LIN {X 0,Y 355.498,Z 368.258,A -85,B 0,C 180,E1 -13423.14,E2 -13423.14} C_VEL
LIN {X 0,Y 356.575,Z 358.586,A -85,B 0,C 180,E1 -13424.845,E2 -13424.845} C_VEL
LIN {X 0,Y 357.7,Z 348.667,A -85,B 0,C 180,E1 -13426.258,E2 -13426.258} C_VEL
LIN {X 0,Y 359.05,Z 337.613,A -85,B 0,C 180,E1 -13427.513,E2 -13427.513} C_VEL
LIN {X 0,Y 359.817,Z 328.864,A -85,B 0,C 180,E1 -13428.335,E2 -13428.335} C_VEL
LIN {X 0,Y 359.129,Z 316.785,A -85,B 0,C 180,E1 -13429.331,E2 -13429.331} C_VEL
LIN {X 0,Y 357.275,Z 303.493,A -85,B 0,C 180,E1 -13430.237,E2 -13430.237} C_VEL
LIN {X 0,Y 354.783,Z 291.013,A -85,B 0,C 180,E1 -13430.922,E2 -13430.922} C_VEL
LIN {X 0,Y 354.186,Z 288.154,A -85,B 0,C 180,E1 -13431.077,E2 -13431.077} C_VEL
LIN {X 0,Y 354.706,Z 281.188,A -85,B 0,C 180,E1 -13434.586,E2 -13434.586} C_VEL
LIN {X 0,Y 355.351,Z 273.981,A -85,B 0,C 180,E1 -13438.336,E2 -13438.336} C_VEL
LIN {X 0,Y 356.313,Z 266.953,A -85,B 0,C 180,E1 -13442.177,E2 -13442.177} C_VEL
LIN {X 0,Y 357.117,Z 261.205,A -85,B 0,C 180,E1 -13445.488,E2 -13445.488} C_VEL
LIN {X 0,Y 357.179,Z 257.764,A -85,B 0,C 180,E1 -13447.586,E2 -13447.586} C_VEL
LIN {X 0,Y 356.457,Z 253.353,A -85,B 0,C 180,E1 -13450.588,E2 -13450.588} C_VEL
LIN {X 0,Y 355.653,Z 249.108,A -85,B 0,C 180,E1 -13453.757,E2 -13453.757} C_VEL
LIN {X 0,Y 354.818,Z 244.397,A -85,B 0,C 180,E1 -13457.664,E2 -13457.664} C_VEL
LIN {X 0,Y 354.814,Z 244.29,A -85,B 0,C 180,E1 -13460.664,E2 -13460.664} C_VEL
LIN {X 0,Y 354.821,Z 244.29,A -85,B 0,C 180,E1 -13464.299,E2 -13464.299} C_VEL
LIN {X 0,Y 354.785,Z 244.294,A -85,B 0,C 180,E1 -13467.665,E2 -13467.665} C_VEL
LIN {X 0,Y 354.867,Z 244.283,A -85,B 0,C 180,E1 -13470.62,E2 -13470.62} C_VEL
LIN {X 0,Y 354.896,Z 244.279,A -85,B 0,C 180,E1 -13474.171,E2 -13474.171} C_VEL
LIN {X 0,Y 354.831,Z 244.287,A -85,B 0,C 180,E1 -13477.892,E2 -13477.892} C_VEL
LIN {X 0,Y 354.919,Z 244.276,A -85,B 0,C 180,E1 -13481.889,E2 -13481.889} C_VEL
LIN {X 0,Y 354.939,Z 244.273,A -85,B 0,C 180,E1 -13485.979,E2 -13485.979} C_VEL
LIN {X 0,Y 354.978,Z 244.269,A -85,B 0,C 180,E1 -13489.734,E2 -13489.734} C_VEL
LIN {X 0,Y 355.109,Z 244.253,A -85,B 0,C 180,E1 -13492.035,E2 -13492.035} C_VEL
LIN {X 0,Y 355.088,Z 244.255,A -85,B 0,C 180,E1 -13494.319,E2 -13494.319} C_VEL
LIN {X 0,Y 355.24,Z 244.237,A -85,B 0,C 180,E1 -13497.731,E2 -13497.731} C_VEL
LIN {X 0,Y 355.391,Z 244.218,A -85,B 0,C 180,E1 -13499.998,E2 -13499.998} C_VEL
LIN {X 0,Y 355.239,Z 244.236,A -85,B 0,C 180,E1 -13502.266,E2 -13502.266} C_VEL
LIN {X 0,Y 355.131,Z 244.248,A -85,B 0,C 180,E1 -13506.817,E2 -13506.817} C_VEL
LIN {X 0,Y 355.009,Z 244.265,A -85,B 0,C 180,E1 -13509.111,E2 -13509.111} C_VEL
LIN {X 0,Y 354.919,Z 244.278,A -85,B 0,C 180,E1 -13512.579,E2 -13512.579} C_VEL
LIN {X 0,Y 354.902,Z 244.283,A -85,B 0,C 180,E1 -13514.916,E2 -13514.916} C_VEL
LIN {X 0,Y 354.68,Z 244.423,A -85,B 0,C 180,E1 -13518.482,E2 -13518.482} C_VEL
LIN {X 0,Y 354.626,Z 246.61,A -85,B 0,C 180,E1 -13521.342,E2 -13521.342} C_VEL
LIN {X 0,Y 354.422,Z 249.207,A -85,B 0,C 180,E1 -13524.606,E2 -13524.606} C_VEL
LIN {X 0,Y 354.268,Z 251.288,A -85,B 0,C 180,E1 -13527.145,E2 -13527.145} C_VEL
LIN {X 0,Y 354.101,Z 254.612,A -85,B 0,C 180,E1 -13531.064,E2 -13531.064} C_VEL
LIN {X 0,Y 354.054,Z 255.479,A -85,B 0,C 180,E1 -13532.06,E2 -13532.06} C_VEL
LIN {X 0,Y 358.257,Z 268.684,A -85,B 0,C 180,E1 -13532.938,E2 -13532.938} C_VEL
LIN {X 0,Y 361.348,Z 281.027,A -85,B 0,C 180,E1 -13533.916,E2 -13533.916} C_VEL
LIN {X 0,Y 361.972,Z 285.048,A -85,B 0,C 180,E1 -13534.265,E2 -13534.265} C_VEL
LIN {X 0,Y 360.855,Z 297.139,A -85,B 0,C 180,E1 -13535.286,E2 -13535.286} C_VEL
LIN {X 0,Y 359.656,Z 308.379,A -85,B 0,C 180,E1 -13536.515,E2 -13536.515} C_VEL
LIN {X 0,Y 358.536,Z 318.063,A -85,B 0,C 180,E1 -13537.834,E2 -13537.834} C_VEL
LIN {X 0,Y 357.357,Z 327.38,A -85,B 0,C 180,E1 -13539.408,E2 -13539.408} C_VEL
LIN {X 0,Y 356.305,Z 334.944,A -85,B 0,C 180,E1 -13540.992,E2 -13540.992} C_VEL
LIN {X 0,Y 355.515,Z 341.121,A -85,B 0,C 180,E1 -13542.587,E2 -13542.587} C_VEL
LIN {X 0,Y 354.693,Z 346.992,A -85,B 0,C 180,E1 -13544.496,E2 -13544.496} C_VEL
LIN {X 0,Y 354.224,Z 350.615,A -85,B 0,C 180,E1 -13546.021,E2 -13546.021} C_VEL
LIN {X 0,Y 353.862,Z 353.392,A -85,B 0,C 180,E1 -13547.527,E2 -13547.527} C_VEL
LIN {X 0,Y 353.531,Z 355.456,A -85,B 0,C 180,E1 -13549.058,E2 -13549.058} C_VEL
LIN {X 0,Y 353.295,Z 356.917,A -85,B 0,C 180,E1 -13550.875,E2 -13550.875} C_VEL
LIN {X 0,Y 353.213,Z 357.364,A -85,B 0,C 180,E1 -13552.736,E2 -13552.736} C_VEL
LIN {X 0,Y 353.253,Z 356.634,A -85,B 0,C 180,E1 -13554.765,E2 -13554.765} C_VEL
LIN {X 0,Y 353.442,Z 354.858,A -85,B 0,C 180,E1 -13556.627,E2 -13556.627} C_VEL
LIN {X 0,Y 353.784,Z 351.63,A -85,B 0,C 180,E1 -13558.667,E2 -13558.667} C_VEL
LIN {X 0,Y 354.247,Z 346.741,A -85,B 0,C 180,E1 -13560.795,E2 -13560.795} C_VEL
LIN {X 0,Y 354.791,Z 341.232,A -85,B 0,C 180,E1 -13562.578,E2 -13562.578} C_VEL
LIN {X 0,Y 355.616,Z 333.637,A -85,B 0,C 180,E1 -13564.503,E2 -13564.503} C_VEL
LIN {X 0,Y 356.492,Z 325.384,A -85,B 0,C 180,E1 -13566.164,E2 -13566.164} C_VEL
LIN {X 0,Y 357.429,Z 316.992,A -85,B 0,C 180,E1 -13567.533,E2 -13567.533} C_VEL
LIN {X 0,Y 358.42,Z 306.878,A -85,B 0,C 180,E1 -13568.882,E2 -13568.882} C_VEL
LIN {X 0,Y 359.467,Z 295.007,A -85,B 0,C 180,E1 -13570.148,E2 -13570.148} C_VEL
LIN {X 0,Y 360.329,Z 282.907,A -85,B 0,C 180,E1 -13571.142,E2 -13571.142} C_VEL
LIN {X 0,Y 359.432,Z 276.737,A -85,B 0,C 180,E1 -13571.619,E2 -13571.619} C_VEL
LIN {X 0,Y 356.469,Z 263.781,A -85,B 0,C 180,E1 -13572.489,E2 -13572.489} C_VEL
LIN {X 0,Y 353.859,Z 253.689,A -85,B 0,C 180,E1 -13573.041,E2 -13573.041} C_VEL
LIN {X 0,Y 354.018,Z 249.56,A -85,B 0,C 180,E1 -13577.388,E2 -13577.388} C_VEL
LIN {X 0,Y 354.153,Z 246.317,A -85,B 0,C 180,E1 -13580.866,E2 -13580.866} C_VEL
LIN {X 0,Y 354.318,Z 244.354,A -85,B 0,C 180,E1 -13583.166,E2 -13583.166} C_VEL
LIN {X 0,Y 354.57,Z 244.321,A -85,B 0,C 180,E1 -13585.454,E2 -13585.454} C_VEL
LIN {X 0,Y 355.132,Z 244.247,A -85,B 0,C 180,E1 -13588.867,E2 -13588.867} C_VEL
LIN {X 0,Y 355.357,Z 244.218,A -85,B 0,C 180,E1 -13590.001,E2 -13590.001} C_VEL
LIN {X 0,Y 355.232,Z 244.233,A -85,B 0,C 180,E1 -13592.269,E2 -13592.269} C_VEL
LIN {X 0,Y 355.124,Z 244.249,A -85,B 0,C 180,E1 -13596.821,E2 -13596.821} C_VEL
LIN {X 0,Y 355.004,Z 244.267,A -85,B 0,C 180,E1 -13599.114,E2 -13599.114} C_VEL
LIN {X 0,Y 354.914,Z 244.274,A -85,B 0,C 180,E1 -13602.582,E2 -13602.582} C_VEL
LIN {X 0,Y 354.878,Z 244.277,A -85,B 0,C 180,E1 -13606.098,E2 -13606.098} C_VEL
LIN {X 0,Y 354.898,Z 244.276,A -85,B 0,C 180,E1 -13608.473,E2 -13608.473} C_VEL
LIN {X 0,Y 354.839,Z 244.282,A -85,B 0,C 180,E1 -13612.107,E2 -13612.107} C_VEL
LIN {X 0,Y 354.889,Z 244.276,A -85,B 0,C 180,E1 -13615.829,E2 -13615.829} C_VEL
LIN {X 0,Y 354.844,Z 244.281,A -85,B 0,C 180,E1 -13619.681,E2 -13619.681} C_VEL
LIN {X 0,Y 354.798,Z 244.287,A -85,B 0,C 180,E1 -13623.704,E2 -13623.704} C_VEL
LIN {X 0,Y 354.792,Z 244.292,A -85,B 0,C 180,E1 -13626.461,E2 -13626.461} C_VEL
LIN {X 0,Y 354.805,Z 244.285,A -85,B 0,C 180,E1 -13629.814,E2 -13629.814} C_VEL
LIN {X 0,Y 354.128,Z 244.375,A -85,B 0,C 180,E1 -13630.761,E2 -13630.761} C_VEL
LIN {X 0,Y 351.245,Z 244.733,A -85,B 0,C 180,E1 -13632.301,E2 -13632.301} C_VEL
LIN {X 0,Y 348.832,Z 245.03,A -85,B 0,C 180,E1 -13633.547,E2 -13633.547} C_VEL
LIN {X 0,Y 347.839,Z 245.159,A -85,B 0,C 180,E1 -13634.512,E2 -13634.512} C_VEL
LIN {X 0,Y 347.78,Z 245.162,A -85,B 0,C 180,E1 -13634.838,E2 -13634.838} C_VEL
LIN {X 0,Y 347.764,Z 245.168,A -85,B 0,C 180,E1 -13638.396,E2 -13638.396} C_VEL
LIN {X 0,Y 347.776,Z 245.164,A -85,B 0,C 180,E1 -13642.013,E2 -13642.013} C_VEL
LIN {X 0,Y 347.742,Z 245.166,A -85,B 0,C 180,E1 -13645.539,E2 -13645.539} C_VEL
LIN {X 0,Y 347.744,Z 245.171,A -85,B 0,C 180,E1 -13648.303,E2 -13648.303} C_VEL
LIN {X 0,Y 347.778,Z 245.162,A -85,B 0,C 180,E1 -13650.99,E2 -13650.99} C_VEL
LIN {X 0,Y 347.831,Z 245.156,A -85,B 0,C 180,E1 -13653.61,E2 -13653.61} C_VEL
LIN {X 0,Y 347.79,Z 245.166,A -85,B 0,C 180,E1 -13656.164,E2 -13656.164} C_VEL
LIN {X 0,Y 347.82,Z 245.16,A -85,B 0,C 180,E1 -13659.912,E2 -13659.912} C_VEL
LIN {X 0,Y 347.87,Z 245.153,A -85,B 0,C 180,E1 -13662.362,E2 -13662.362} C_VEL
LIN {X 0,Y 347.902,Z 245.151,A -85,B 0,C 180,E1 -13665.973,E2 -13665.973} C_VEL
LIN {X 0,Y 347.935,Z 245.144,A -85,B 0,C 180,E1 -13669.528,E2 -13669.528} C_VEL
LIN {X 0,Y 348.084,Z 245.124,A -85,B 0,C 180,E1 -13673.044,E2 -13673.044} C_VEL
LIN {X 0,Y 348.212,Z 245.112,A -85,B 0,C 180,E1 -13677.688,E2 -13677.688} C_VEL
LIN {X 0,Y 348.332,Z 245.096,A -85,B 0,C 180,E1 -13680.002,E2 -13680.002} C_VEL
LIN {X 0,Y 348.21,Z 245.109,A -85,B 0,C 180,E1 -13682.315,E2 -13682.315} C_VEL
LIN {X 0,Y 348.085,Z 245.124,A -85,B 0,C 180,E1 -13686.96,E2 -13686.96} C_VEL
LIN {X 0,Y 347.905,Z 245.146,A -85,B 0,C 180,E1 -13690.477,E2 -13690.477} C_VEL
LIN {X 0,Y 347.908,Z 245.146,A -85,B 0,C 180,E1 -13694.151,E2 -13694.151} C_VEL
LIN {X 0,Y 347.9,Z 245.146,A -85,B 0,C 180,E1 -13698.291,E2 -13698.291} C_VEL
LIN {X 0,Y 347.797,Z 245.163,A -85,B 0,C 180,E1 -13701.635,E2 -13701.635} C_VEL
LIN {X 0,Y 347.822,Z 245.16,A -85,B 0,C 180,E1 -13705.109,E2 -13705.109} C_VEL
LIN {X 0,Y 347.818,Z 245.159,A -85,B 0,C 180,E1 -13707.695,E2 -13707.695} C_VEL
LIN {X 0,Y 347.759,Z 245.164,A -85,B 0,C 180,E1 -13710.349,E2 -13710.349} C_VEL
LIN {X 0,Y 347.758,Z 245.164,A -85,B 0,C 180,E1 -13714.044,E2 -13714.044} C_VEL
LIN {X 0,Y 347.771,Z 245.166,A -85,B 0,C 180,E1 -13717.321,E2 -13717.321} C_VEL
LIN {X 0,Y 347.742,Z 245.17,A -85,B 0,C 180,E1 -13720.297,E2 -13720.297} C_VEL
LIN {X 0,Y 347.733,Z 245.171,A -85,B 0,C 180,E1 -13723.408,E2 -13723.408} C_VEL
LIN {X 0,Y 347.807,Z 245.271,A -85,B 0,C 180,E1 -13724.604,E2 -13724.604} C_VEL
LIN {X 0,Y 348.803,Z 250.669,A -85,B 0,C 180,E1 -13728.205,E2 -13728.205} C_VEL
LIN {X 0,Y 349.682,Z 256.107,A -85,B 0,C 180,E1 -13731.615,E2 -13731.615} C_VEL
LIN {X 0,Y 349.999,Z 259.154,A -85,B 0,C 180,E1 -13733.439,E2 -13733.439} C_VEL
LIN {X 0,Y 349.634,Z 263.233,A -85,B 0,C 180,E1 -13735.747,E2 -13735.747} C_VEL
LIN {X 0,Y 348.836,Z 269.351,A -85,B 0,C 180,E1 -13739.085,E2 -13739.085} C_VEL
LIN {X 0,Y 348.079,Z 276.104,A -85,B 0,C 180,E1 -13742.675,E2 -13742.675} C_VEL
LIN {X 0,Y 347.485,Z 282.774,A -85,B 0,C 180,E1 -13746.139,E2 -13746.139} C_VEL
LIN {X 0,Y 346.999,Z 289.61,A -85,B 0,C 180,E1 -13749.588,E2 -13749.588} C_VEL
LIN {X 0,Y 349.211,Z 303.34,A -85,B 0,C 180,E1 -13750.216,E2 -13750.216} C_VEL
LIN {X 0,Y 350.795,Z 315.397,A -85,B 0,C 180,E1 -13750.977,E2 -13750.977} C_VEL
LIN {X 0,Y 351.821,Z 327.79,A -85,B 0,C 180,E1 -13751.962,E2 -13751.962} C_VEL
LIN {X 0,Y 351.492,Z 334.288,A -85,B 0,C 180,E1 -13752.546,E2 -13752.546} C_VEL
LIN {X 0,Y 350.348,Z 345,A -85,B 0,C 180,E1 -13753.688,E2 -13753.688} C_VEL
LIN {X 0,Y 349.248,Z 355.917,A -85,B 0,C 180,E1 -13755.154,E2 -13755.154} C_VEL
LIN {X 0,Y 348.324,Z 364.544,A -85,B 0,C 180,E1 -13756.582,E2 -13756.582} C_VEL
LIN {X 0,Y 347.622,Z 371.791,A -85,B 0,C 180,E1 -13758.039,E2 -13758.039} C_VEL
LIN {X 0,Y 346.938,Z 378.901,A -85,B 0,C 180,E1 -13759.789,E2 -13759.789} C_VEL
LIN {X 0,Y 346.495,Z 385.391,A -85,B 0,C 180,E1 -13761.836,E2 -13761.836} C_VEL
LIN {X 0,Y 346.304,Z 389.782,A -85,B 0,C 180,E1 -13763.649,E2 -13763.649} C_VEL
LIN {X 0,Y 346.257,Z 392.837,A -85,B 0,C 180,E1 -13765.342,E2 -13765.342} C_VEL
LIN {X 0,Y 346.226,Z 394.407,A -85,B 0,C 180,E1 -13766.508,E2 -13766.508} C_VEL
LIN {X 0,Y 346.277,Z 395.549,A -85,B 0,C 180,E1 -13767.672,E2 -13767.672} C_VEL
LIN {X 0,Y 346.384,Z 396.25,A -85,B 0,C 180,E1 -13768.836,E2 -13768.836} C_VEL
LIN {X 0,Y 346.389,Z 396.548,A -85,B 0,C 180,E1 -13769.999,E2 -13769.999} C_VEL
LIN {X 0,Y 346.357,Z 396.449,A -85,B 0,C 180,E1 -13771.162,E2 -13771.162} C_VEL
LIN {X 0,Y 346.247,Z 395.936,A -85,B 0,C 180,E1 -13772.325,E2 -13772.325} C_VEL
LIN {X 0,Y 346.205,Z 394.987,A -85,B 0,C 180,E1 -13773.49,E2 -13773.49} C_VEL
LIN {X 0,Y 346.227,Z 393.638,A -85,B 0,C 180,E1 -13774.656,E2 -13774.656} C_VEL
LIN {X 0,Y 346.285,Z 390.811,A -85,B 0,C 180,E1 -13776.407,E2 -13776.407} C_VEL
LIN {X 0,Y 346.495,Z 386.957,A -85,B 0,C 180,E1 -13778.161,E2 -13778.161} C_VEL
LIN {X 0,Y 346.885,Z 381.991,A -85,B 0,C 180,E1 -13779.915,E2 -13779.915} C_VEL
LIN {X 0,Y 347.487,Z 375.766,A -85,B 0,C 180,E1 -13781.667,E2 -13781.667} C_VEL
LIN {X 0,Y 348.563,Z 368.076,A -85,B 0,C 180,E1 -13783.406,E2 -13783.406} C_VEL
LIN {X 0,Y 349.486,Z 360.249,A -85,B 0,C 180,E1 -13784.855,E2 -13784.855} C_VEL
LIN {X 0,Y 350.593,Z 350.749,A -85,B 0,C 180,E1 -13786.297,E2 -13786.297} C_VEL
LIN {X 0,Y 351.946,Z 340.283,A -85,B 0,C 180,E1 -13787.578,E2 -13787.578} C_VEL
LIN {X 0,Y 353.03,Z 330.307,A -85,B 0,C 180,E1 -13788.572,E2 -13788.572} C_VEL
LIN {X 0,Y 352.496,Z 318.922,A -85,B 0,C 180,E1 -13789.575,E2 -13789.575} C_VEL
LIN {X 0,Y 350.891,Z 306.196,A -85,B 0,C 180,E1 -13790.515,E2 -13790.515} C_VEL
LIN {X 0,Y 348.426,Z 293.291,A -85,B 0,C 180,E1 -13791.288,E2 -13791.288} C_VEL
LIN {X 0,Y 347.159,Z 287.71,A -85,B 0,C 180,E1 -13791.605,E2 -13791.605} C_VEL
LIN {X 0,Y 347.731,Z 280.924,A -85,B 0,C 180,E1 -13795.113,E2 -13795.113} C_VEL
LIN {X 0,Y 348.43,Z 273.782,A -85,B 0,C 180,E1 -13798.952,E2 -13798.952} C_VEL
LIN {X 0,Y 349.305,Z 267.767,A -85,B 0,C 180,E1 -13802.322,E2 -13802.322} C_VEL
LIN {X 0,Y 350.128,Z 262.199,A -85,B 0,C 180,E1 -13805.597,E2 -13805.597} C_VEL
LIN {X 0,Y 350.201,Z 258.858,A -85,B 0,C 180,E1 -13807.721,E2 -13807.721} C_VEL
LIN {X 0,Y 349.59,Z 255.275,A -85,B 0,C 180,E1 -13810.186,E2 -13810.186} C_VEL
LIN {X 0,Y 348.757,Z 250.896,A -85,B 0,C 180,E1 -13813.491,E2 -13813.491} C_VEL
LIN {X 0,Y 348.103,Z 247.088,A -85,B 0,C 180,E1 -13816.649,E2 -13816.649} C_VEL
LIN {X 0,Y 347.756,Z 245.169,A -85,B 0,C 180,E1 -13818.394,E2 -13818.394} C_VEL
LIN {X 0,Y 347.773,Z 245.168,A -85,B 0,C 180,E1 -13822.009,E2 -13822.009} C_VEL
LIN {X 0,Y 347.743,Z 245.172,A -85,B 0,C 180,E1 -13825.534,E2 -13825.534} C_VEL
LIN {X 0,Y 347.762,Z 245.168,A -85,B 0,C 180,E1 -13829.652,E2 -13829.652} C_VEL
LIN {X 0,Y 347.848,Z 245.158,A -85,B 0,C 180,E1 -13832.743,E2 -13832.743} C_VEL
LIN {X 0,Y 347.785,Z 245.165,A -85,B 0,C 180,E1 -13836.16,E2 -13836.16} C_VEL
LIN {X 0,Y 347.814,Z 245.161,A -85,B 0,C 180,E1 -13839.908,E2 -13839.908} C_VEL
LIN {X 0,Y 347.863,Z 245.155,A -85,B 0,C 180,E1 -13842.357,E2 -13842.357} C_VEL
LIN {X 0,Y 347.893,Z 245.151,A -85,B 0,C 180,E1 -13845.969,E2 -13845.969} C_VEL
LIN {X 0,Y 347.928,Z 245.148,A -85,B 0,C 180,E1 -13849.524,E2 -13849.524} C_VEL
LIN {X 0,Y 348.069,Z 245.13,A -85,B 0,C 180,E1 -13851.873,E2 -13851.873} C_VEL
LIN {X 0,Y 348.063,Z 245.13,A -85,B 0,C 180,E1 -13854.204,E2 -13854.204} C_VEL
LIN {X 0,Y 348.203,Z 245.113,A -85,B 0,C 180,E1 -13857.685,E2 -13857.685} C_VEL
LIN {X 0,Y 348.361,Z 245.093,A -85,B 0,C 180,E1 -13859.998,E2 -13859.998} C_VEL
LIN {X 0,Y 348.202,Z 245.113,A -85,B 0,C 180,E1 -13862.312,E2 -13862.312} C_VEL
LIN {X 0,Y 348.099,Z 245.124,A -85,B 0,C 180,E1 -13866.956,E2 -13866.956} C_VEL
LIN {X 0,Y 347.961,Z 245.143,A -85,B 0,C 180,E1 -13869.297,E2 -13869.297} C_VEL
LIN {X 0,Y 347.885,Z 245.154,A -85,B 0,C 180,E1 -13872.838,E2 -13872.838} C_VEL
LIN {X 0,Y 347.842,Z 245.163,A -85,B 0,C 180,E1 -13875.226,E2 -13875.226} C_VEL
LIN {X 0,Y 347.694,Z 245.306,A -85,B 0,C 180,E1 -13878.195,E2 -13878.195} C_VEL
LIN {X 0,Y 347.572,Z 247.815,A -85,B 0,C 180,E1 -13881.548,E2 -13881.548} C_VEL
LIN {X 0,Y 347.331,Z 250.642,A -85,B 0,C 180,E1 -13885.143,E2 -13885.143} C_VEL
LIN {X 0,Y 347.186,Z 252.758,A -85,B 0,C 180,E1 -13887.745,E2 -13887.745} C_VEL
LIN {X 0,Y 347.048,Z 255.97,A -85,B 0,C 180,E1 -13891.547,E2 -13891.547} C_VEL
LIN {X 0,Y 350.907,Z 267.745,A -85,B 0,C 180,E1 -13892.35,E2 -13892.35} C_VEL
LIN {X 0,Y 353.938,Z 279.056,A -85,B 0,C 180,E1 -13893.264,E2 -13893.264} C_VEL
LIN {X 0,Y 355.291,Z 286.608,A -85,B 0,C 180,E1 -13893.937,E2 -13893.937} C_VEL
LIN {X 0,Y 354.147,Z 298.038,A -85,B 0,C 180,E1 -13894.941,E2 -13894.941} C_VEL
LIN {X 0,Y 352.891,Z 309.313,A -85,B 0,C 180,E1 -13896.207,E2 -13896.207} C_VEL
LIN {X 0,Y 351.705,Z 319.043,A -85,B 0,C 180,E1 -13897.57,E2 -13897.57} C_VEL
LIN {X 0,Y 350.584,Z 327.358,A -85,B 0,C 180,E1 -13899.001,E2 -13899.001} C_VEL
LIN {X 0,Y 349.494,Z 334.949,A -85,B 0,C 180,E1 -13900.604,E2 -13900.604} C_VEL
LIN {X 0,Y 348.448,Z 342.447,A -85,B 0,C 180,E1 -13902.595,E2 -13902.595} C_VEL
LIN {X 0,Y 347.764,Z 347.094,A -85,B 0,C 180,E1 -13904.16,E2 -13904.16} C_VEL
LIN {X 0,Y 347.224,Z 350.92,A -85,B 0,C 180,E1 -13905.779,E2 -13905.779} C_VEL
LIN {X 0,Y 346.659,Z 354.751,A -85,B 0,C 180,E1 -13908.01,E2 -13908.01} C_VEL
LIN {X 0,Y 346.362,Z 356.406,A -85,B 0,C 180,E1 -13909.512,E2 -13909.512} C_VEL
LIN {X 0,Y 346.196,Z 357.41,A -85,B 0,C 180,E1 -13911.002,E2 -13911.002} C_VEL
LIN {X 0,Y 346.128,Z 357.754,A -85,B 0,C 180,E1 -13912.474,E2 -13912.474} C_VEL
LIN {X 0,Y 346.148,Z 357.298,A -85,B 0,C 180,E1 -13914.301,E2 -13914.301} C_VEL
LIN {X 0,Y 346.294,Z 355.68,A -85,B 0,C 180,E1 -13916.31,E2 -13916.31} C_VEL
LIN {X 0,Y 346.648,Z 352.708,A -85,B 0,C 180,E1 -13918.372,E2 -13918.372} C_VEL
LIN {X 0,Y 347.101,Z 348.098,A -85,B 0,C 180,E1 -13920.529,E2 -13920.529} C_VEL
LIN {X 0,Y 347.62,Z 343.068,A -85,B 0,C 180,E1 -13922.291,E2 -13922.291} C_VEL
LIN {X 0,Y 348.302,Z 337.044,A -85,B 0,C 180,E1 -13923.97,E2 -13923.97} C_VEL
LIN {X 0,Y 349.115,Z 329.695,A -85,B 0,C 180,E1 -13925.628,E2 -13925.628} C_VEL
LIN {X 0,Y 350.102,Z 321.112,A -85,B 0,C 180,E1 -13927.189,E2 -13927.189} C_VEL
LIN {X 0,Y 351.215,Z 310.597,A -85,B 0,C 180,E1 -13928.736,E2 -13928.736} C_VEL
LIN {X 0,Y 352.31,Z 299.509,A -85,B 0,C 180,E1 -13930.03,E2 -13930.03} C_VEL
LIN {X 0,Y 353.267,Z 287.417,A -85,B 0,C 180,E1 -13931.14,E2 -13931.14} C_VEL
LIN {X 0,Y 353.514,Z 283.343,A -85,B 0,C 180,E1 -13931.454,E2 -13931.454} C_VEL
LIN {X 0,Y 351.416,Z 272.528,A -85,B 0,C 180,E1 -13932.295,E2 -13932.295} C_VEL
LIN {X 0,Y 348.273,Z 259.692,A -85,B 0,C 180,E1 -13933.101,E2 -13933.101} C_VEL
LIN {X 0,Y 346.762,Z 254.07,A -85,B 0,C 180,E1 -13933.404,E2 -13933.404} C_VEL
LIN {X 0,Y 346.935,Z 250.563,A -85,B 0,C 180,E1 -13937.126,E2 -13937.126} C_VEL
LIN {X 0,Y 347.091,Z 247.296,A -85,B 0,C 180,E1 -13940.679,E2 -13940.679} C_VEL
LIN {X 0,Y 347.267,Z 245.233,A -85,B 0,C 180,E1 -13943.027,E2 -13943.027} C_VEL
LIN {X 0,Y 347.527,Z 245.198,A -85,B 0,C 180,E1 -13945.361,E2 -13945.361} C_VEL
LIN {X 0,Y 348.094,Z 245.123,A -85,B 0,C 180,E1 -13948.844,E2 -13948.844} C_VEL
LIN {X 0,Y 348.306,Z 245.097,A -85,B 0,C 180,E1 -13950.001,E2 -13950.001} C_VEL
LIN {X 0,Y 348.195,Z 245.109,A -85,B 0,C 180,E1 -13952.315,E2 -13952.315} C_VEL
LIN {X 0,Y 348.092,Z 245.126,A -85,B 0,C 180,E1 -13956.959,E2 -13956.959} C_VEL
LIN {X 0,Y 347.956,Z 245.144,A -85,B 0,C 180,E1 -13959.3,E2 -13959.3} C_VEL
LIN {X 0,Y 347.882,Z 245.152,A -85,B 0,C 180,E1 -13962.841,E2 -13962.841} C_VEL
LIN {X 0,Y 347.827,Z 245.156,A -85,B 0,C 180,E1 -13966.433,E2 -13966.433} C_VEL
LIN {X 0,Y 347.85,Z 245.157,A -85,B 0,C 180,E1 -13968.862,E2 -13968.862} C_VEL
LIN {X 0,Y 347.802,Z 245.159,A -85,B 0,C 180,E1 -13971.647,E2 -13971.647} C_VEL
LIN {X 0,Y 347.807,Z 245.162,A -85,B 0,C 180,E1 -13975.11,E2 -13975.11} C_VEL
LIN {X 0,Y 347.8,Z 245.159,A -85,B 0,C 180,E1 -13977.696,E2 -13977.696} C_VEL
LIN {X 0,Y 347.755,Z 245.166,A -85,B 0,C 180,E1 -13980.349,E2 -13980.349} C_VEL
LIN {X 0,Y 347.736,Z 245.17,A -85,B 0,C 180,E1 -13984.466,E2 -13984.466} C_VEL
LIN {X 0,Y 347.769,Z 245.163,A -85,B 0,C 180,E1 -13987.992,E2 -13987.992} C_VEL
LIN {X 0,Y 347.778,Z 245.162,A -85,B 0,C 180,E1 -13991.611,E2 -13991.611} C_VEL
LIN {X 0,Y 347.78,Z 245.162,A -85,B 0,C 180,E1 -13994.838,E2 -13994.838} C_VEL
LIN {X 0,Y 347.165,Z 245.244,A -85,B 0,C 180,E1 -13995.805,E2 -13995.805} C_VEL
LIN {X 0,Y 344.303,Z 245.599,A -85,B 0,C 180,E1 -13997.377,E2 -13997.377} C_VEL
LIN {X 0,Y 341.843,Z 245.905,A -85,B 0,C 180,E1 -13998.65,E2 -13998.65} C_VEL
LIN {X 0,Y 340.787,Z 246.033,A -85,B 0,C 180,E1 -13999.636,E2 -13999.636} C_VEL
LIN {X 0,Y 340.703,Z 246.044,A -85,B 0,C 180,E1 -13999.97,E2 -13999.97} C_VEL
LIN {X 0,Y 340.709,Z 246.042,A -85,B 0,C 180,E1 -14003.561,E2 -14003.561} C_VEL
LIN {X 0,Y 340.691,Z 246.048,A -85,B 0,C 180,E1 -14006.156,E2 -14006.156} C_VEL
LIN {X 0,Y 340.741,Z 246.043,A -85,B 0,C 180,E1 -14010.332,E2 -14010.332} C_VEL
LIN {X 0,Y 340.803,Z 246.03,A -85,B 0,C 180,E1 -14013.022,E2 -14013.022} C_VEL
LIN {X 0,Y 340.73,Z 246.04,A -85,B 0,C 180,E1 -14016.93,E2 -14016.93} C_VEL
LIN {X 0,Y 340.797,Z 246.032,A -85,B 0,C 180,E1 -14020.736,E2 -14020.736} C_VEL
LIN {X 0,Y 340.79,Z 246.032,A -85,B 0,C 180,E1 -14023.221,E2 -14023.221} C_VEL
LIN {X 0,Y 340.851,Z 246.024,A -85,B 0,C 180,E1 -14026.893,E2 -14026.893} C_VEL
LIN {X 0,Y 340.917,Z 246.017,A -85,B 0,C 180,E1 -14030.509,E2 -14030.509} C_VEL
LIN {X 0,Y 341.051,Z 245.999,A -85,B 0,C 180,E1 -14032.9,E2 -14032.9} C_VEL
LIN {X 0,Y 341.173,Z 245.988,A -85,B 0,C 180,E1 -14037.641,E2 -14037.641} C_VEL
LIN {X 0,Y 341.283,Z 245.974,A -85,B 0,C 180,E1 -14040.002,E2 -14040.002} C_VEL
LIN {X 0,Y 341.172,Z 245.985,A -85,B 0,C 180,E1 -14042.363,E2 -14042.363} C_VEL
LIN {X 0,Y 341.053,Z 246,A -85,B 0,C 180,E1 -14047.104,E2 -14047.104} C_VEL
LIN {X 0,Y 340.856,Z 246.024,A -85,B 0,C 180,E1 -14050.696,E2 -14050.696} C_VEL
LIN {X 0,Y 340.872,Z 246.022,A -85,B 0,C 180,E1 -14054.326,E2 -14054.326} C_VEL
LIN {X 0,Y 340.846,Z 246.025,A -85,B 0,C 180,E1 -14058.467,E2 -14058.467} C_VEL
LIN {X 0,Y 340.764,Z 246.037,A -85,B 0,C 180,E1 -14061.858,E2 -14061.858} C_VEL
LIN {X 0,Y 340.782,Z 246.035,A -85,B 0,C 180,E1 -14065.665,E2 -14065.665} C_VEL
LIN {X 0,Y 340.738,Z 246.038,A -85,B 0,C 180,E1 -14068.322,E2 -14068.322} C_VEL
LIN {X 0,Y 340.708,Z 246.046,A -85,B 0,C 180,E1 -14071.045,E2 -14071.045} C_VEL
LIN {X 0,Y 340.728,Z 246.044,A -85,B 0,C 180,E1 -14075.279,E2 -14075.279} C_VEL
LIN {X 0,Y 340.719,Z 246.041,A -85,B 0,C 180,E1 -14078.386,E2 -14078.386} C_VEL
LIN {X 0,Y 340.709,Z 246.046,A -85,B 0,C 180,E1 -14082.046,E2 -14082.046} C_VEL
LIN {X 0,Y 340.743,Z 246.199,A -85,B 0,C 180,E1 -14084.315,E2 -14084.315} C_VEL
LIN {X 0,Y 341.701,Z 251.247,A -85,B 0,C 180,E1 -14087.771,E2 -14087.771} C_VEL
LIN {X 0,Y 342.571,Z 256.608,A -85,B 0,C 180,E1 -14091.225,E2 -14091.225} C_VEL
LIN {X 0,Y 342.959,Z 260.372,A -85,B 0,C 180,E1 -14093.538,E2 -14093.538} C_VEL
LIN {X 0,Y 342.592,Z 264.179,A -85,B 0,C 180,E1 -14095.727,E2 -14095.727} C_VEL
LIN {X 0,Y 341.792,Z 270.144,A -85,B 0,C 180,E1 -14099.064,E2 -14099.064} C_VEL
LIN {X 0,Y 340.92,Z 277.472,A -85,B 0,C 180,E1 -14103.029,E2 -14103.029} C_VEL
LIN {X 0,Y 340.383,Z 283.542,A -85,B 0,C 180,E1 -14106.256,E2 -14106.256} C_VEL
LIN {X 0,Y 339.96,Z 289.367,A -85,B 0,C 180,E1 -14109.212,E2 -14109.212} C_VEL
LIN {X 0,Y 342.16,Z 302.821,A -85,B 0,C 180,E1 -14109.846,E2 -14109.846} C_VEL
LIN {X 0,Y 343.862,Z 315.773,A -85,B 0,C 180,E1 -14110.687,E2 -14110.687} C_VEL
LIN {X 0,Y 344.914,Z 328.582,A -85,B 0,C 180,E1 -14111.742,E2 -14111.742} C_VEL
LIN {X 0,Y 344.532,Z 334.888,A -85,B 0,C 180,E1 -14112.335,E2 -14112.335} C_VEL
LIN {X 0,Y 343.167,Z 346.572,A -85,B 0,C 180,E1 -14113.643,E2 -14113.643} C_VEL
LIN {X 0,Y 342.214,Z 356.262,A -85,B 0,C 180,E1 -14115.004,E2 -14115.004} C_VEL
LIN {X 0,Y 341.21,Z 365.465,A -85,B 0,C 180,E1 -14116.6,E2 -14116.6} C_VEL
LIN {X 0,Y 340.307,Z 373.726,A -85,B 0,C 180,E1 -14118.383,E2 -14118.383} C_VEL
LIN {X 0,Y 339.759,Z 380.386,A -85,B 0,C 180,E1 -14120.173,E2 -14120.173} C_VEL
LIN {X 0,Y 339.354,Z 386.442,A -85,B 0,C 180,E1 -14122.262,E2 -14122.262} C_VEL
LIN {X 0,Y 339.146,Z 391.154,A -85,B 0,C 180,E1 -14124.494,E2 -14124.494} C_VEL
LIN {X 0,Y 339.147,Z 393.955,A -85,B 0,C 180,E1 -14126.435,E2 -14126.435} C_VEL
LIN {X 0,Y 339.181,Z 395.118,A -85,B 0,C 180,E1 -14127.624,E2 -14127.624} C_VEL
LIN {X 0,Y 339.302,Z 395.832,A -85,B 0,C 180,E1 -14128.812,E2 -14128.812} C_VEL
LIN {X 0,Y 339.328,Z 396.142,A -85,B 0,C 180,E1 -14129.999,E2 -14129.999} C_VEL
LIN {X 0,Y 339.262,Z 396.052,A -85,B 0,C 180,E1 -14131.186,E2 -14131.186} C_VEL
LIN {X 0,Y 339.15,Z 395.558,A -85,B 0,C 180,E1 -14132.374,E2 -14132.374} C_VEL
LIN {X 0,Y 339.127,Z 394.625,A -85,B 0,C 180,E1 -14133.563,E2 -14133.563} C_VEL
LIN {X 0,Y 339.139,Z 391.635,A -85,B 0,C 180,E1 -14135.888,E2 -14135.888} C_VEL
LIN {X 0,Y 339.353,Z 388.069,A -85,B 0,C 180,E1 -14137.735,E2 -14137.735} C_VEL
LIN {X 0,Y 339.684,Z 383.517,A -85,B 0,C 180,E1 -14139.526,E2 -14139.526} C_VEL
LIN {X 0,Y 340.379,Z 376.679,A -85,B 0,C 180,E1 -14141.613,E2 -14141.613} C_VEL
LIN {X 0,Y 341.442,Z 369.264,A -85,B 0,C 180,E1 -14143.388,E2 -14143.388} C_VEL
LIN {X 0,Y 342.502,Z 360.878,A -85,B 0,C 180,E1 -14145.023,E2 -14145.023} C_VEL
LIN {X 0,Y 343.629,Z 351.729,A -85,B 0,C 180,E1 -14146.484,E2 -14146.484} C_VEL
LIN {X 0,Y 344.998,Z 341.595,A -85,B 0,C 180,E1 -14147.791,E2 -14147.791} C_VEL
LIN {X 0,Y 346.212,Z 332.024,A -85,B 0,C 180,E1 -14148.798,E2 -14148.798} C_VEL
LIN {X 0,Y 345.872,Z 321.006,A -85,B 0,C 180,E1 -14149.828,E2 -14149.828} C_VEL
LIN {X 0,Y 344.557,Z 309.259,A -85,B 0,C 180,E1 -14150.763,E2 -14150.763} C_VEL
LIN {X 0,Y 342.266,Z 296.228,A -85,B 0,C 180,E1 -14151.621,E2 -14151.621} C_VEL
LIN {X 0,Y 340.158,Z 287.326,A -85,B 0,C 180,E1 -14152.119,E2 -14152.119} C_VEL
LIN {X 0,Y 340.881,Z 279.475,A -85,B 0,C 180,E1 -14156.311,E2 -14156.311} C_VEL
LIN {X 0,Y 341.7,Z 272.411,A -85,B 0,C 180,E1 -14160.247,E2 -14160.247} C_VEL
LIN {X 0,Y 342.588,Z 266.633,A -85,B 0,C 180,E1 -14163.633,E2 -14163.633} C_VEL
LIN {X 0,Y 343.205,Z 262.071,A -85,B 0,C 180,E1 -14166.429,E2 -14166.429} C_VEL
LIN {X 0,Y 343.179,Z 259.849,A -85,B 0,C 180,E1 -14167.905,E2 -14167.905} C_VEL
LIN {X 0,Y 342.397,Z 255.466,A -85,B 0,C 180,E1 -14171.057,E2 -14171.057} C_VEL
LIN {X 0,Y 341.574,Z 251.225,A -85,B 0,C 180,E1 -14174.39,E2 -14174.39} C_VEL
LIN {X 0,Y 340.884,Z 247.212,A -85,B 0,C 180,E1 -14177.918,E2 -14177.918} C_VEL
LIN {X 0,Y 340.69,Z 246.05,A -85,B 0,C 180,E1 -14179.126,E2 -14179.126} C_VEL
LIN {X 0,Y 340.732,Z 246.045,A -85,B 0,C 180,E1 -14181.771,E2 -14181.771} C_VEL
LIN {X 0,Y 340.721,Z 246.047,A -85,B 0,C 180,E1 -14185.594,E2 -14185.594} C_VEL
LIN {X 0,Y 340.702,Z 246.049,A -85,B 0,C 180,E1 -14188.954,E2 -14188.954} C_VEL
LIN {X 0,Y 340.775,Z 246.039,A -85,B 0,C 180,E1 -14192.473,E2 -14192.473} C_VEL
LIN {X 0,Y 340.753,Z 246.041,A -85,B 0,C 180,E1 -14195.636,E2 -14195.636} C_VEL
LIN {X 0,Y 340.745,Z 246.042,A -85,B 0,C 180,E1 -14199.472,E2 -14199.472} C_VEL
LIN {X 0,Y 340.854,Z 246.028,A -85,B 0,C 180,E1 -14201.982,E2 -14201.982} C_VEL
LIN {X 0,Y 340.865,Z 246.026,A -85,B 0,C 180,E1 -14205.703,E2 -14205.703} C_VEL
LIN {X 0,Y 340.87,Z 246.027,A -85,B 0,C 180,E1 -14209.304,E2 -14209.304} C_VEL
LIN {X 0,Y 341.07,Z 246.001,A -85,B 0,C 180,E1 -14212.896,E2 -14212.896} C_VEL
LIN {X 0,Y 341.164,Z 245.99,A -85,B 0,C 180,E1 -14217.637,E2 -14217.637} C_VEL
LIN {X 0,Y 341.309,Z 245.972,A -85,B 0,C 180,E1 -14219.998,E2 -14219.998} C_VEL
LIN {X 0,Y 341.164,Z 245.99,A -85,B 0,C 180,E1 -14222.359,E2 -14222.359} C_VEL
LIN {X 0,Y 341.068,Z 245.999,A -85,B 0,C 180,E1 -14227.1,E2 -14227.1} C_VEL
LIN {X 0,Y 340.868,Z 246.026,A -85,B 0,C 180,E1 -14230.692,E2 -14230.692} C_VEL
LIN {X 0,Y 340.853,Z 246.032,A -85,B 0,C 180,E1 -14234.323,E2 -14234.323} C_VEL
LIN {X 0,Y 340.687,Z 246.287,A -85,B 0,C 180,E1 -14238.023,E2 -14238.023} C_VEL
LIN {X 0,Y 340.534,Z 249.062,A -85,B 0,C 180,E1 -14241.805,E2 -14241.805} C_VEL
LIN {X 0,Y 340.353,Z 251.263,A -85,B 0,C 180,E1 -14244.696,E2 -14244.696} C_VEL
LIN {X 0,Y 340.124,Z 254.218,A -85,B 0,C 180,E1 -14248.373,E2 -14248.373} C_VEL
LIN {X 0,Y 340.013,Z 256.368,A -85,B 0,C 180,E1 -14250.993,E2 -14250.993} C_VEL
LIN {X 0,Y 344.757,Z 270.758,A -85,B 0,C 180,E1 -14252.047,E2 -14252.047} C_VEL
LIN {X 0,Y 347.773,Z 282.554,A -85,B 0,C 180,E1 -14253.065,E2 -14253.065} C_VEL
LIN {X 0,Y 348.648,Z 287.976,A -85,B 0,C 180,E1 -14253.576,E2 -14253.576} C_VEL
LIN {X 0,Y 347.464,Z 299.19,A -85,B 0,C 180,E1 -14254.6,E2 -14254.6} C_VEL
LIN {X 0,Y 346.17,Z 310.016,A -85,B 0,C 180,E1 -14255.851,E2 -14255.851} C_VEL
LIN {X 0,Y 344.83,Z 320.408,A -85,B 0,C 180,E1 -14257.36,E2 -14257.36} C_VEL
LIN {X 0,Y 343.546,Z 329.332,A -85,B 0,C 180,E1 -14258.981,E2 -14258.981} C_VEL
LIN {X 0,Y 342.428,Z 336.561,A -85,B 0,C 180,E1 -14260.592,E2 -14260.592} C_VEL
LIN {X 0,Y 341.557,Z 342.453,A -85,B 0,C 180,E1 -14262.207,E2 -14262.207} C_VEL
LIN {X 0,Y 340.853,Z 347.198,A -85,B 0,C 180,E1 -14263.81,E2 -14263.81} C_VEL
LIN {X 0,Y 340.271,Z 350.959,A -85,B 0,C 180,E1 -14265.395,E2 -14265.395} C_VEL
LIN {X 0,Y 339.829,Z 353.867,A -85,B 0,C 180,E1 -14266.965,E2 -14266.965} C_VEL
LIN {X 0,Y 339.473,Z 355.943,A -85,B 0,C 180,E1 -14268.512,E2 -14268.512} C_VEL
LIN {X 0,Y 339.226,Z 357.324,A -85,B 0,C 180,E1 -14270.042,E2 -14270.042} C_VEL
LIN {X 0,Y 339.064,Z 358.116,A -85,B 0,C 180,E1 -14271.963,E2 -14271.963} C_VEL
LIN {X 0,Y 339.042,Z 357.85,A -85,B 0,C 180,E1 -14273.939,E2 -14273.939} C_VEL
LIN {X 0,Y 339.186,Z 356.415,A -85,B 0,C 180,E1 -14275.984,E2 -14275.984} C_VEL
LIN {X 0,Y 339.499,Z 353.709,A -85,B 0,C 180,E1 -14278.071,E2 -14278.071} C_VEL
LIN {X 0,Y 339.97,Z 349.407,A -85,B 0,C 180,E1 -14280.257,E2 -14280.257} C_VEL
LIN {X 0,Y 340.503,Z 344.371,A -85,B 0,C 180,E1 -14282.136,E2 -14282.136} C_VEL
LIN {X 0,Y 341.246,Z 337.803,A -85,B 0,C 180,E1 -14284.048,E2 -14284.048} C_VEL
LIN {X 0,Y 342.077,Z 330.538,A -85,B 0,C 180,E1 -14285.74,E2 -14285.74} C_VEL
LIN {X 0,Y 343.183,Z 321.17,A -85,B 0,C 180,E1 -14287.483,E2 -14287.483} C_VEL
LIN {X 0,Y 344.263,Z 311.639,A -85,B 0,C 180,E1 -14288.913,E2 -14288.913} C_VEL
LIN {X 0,Y 345.387,Z 300.795,A -85,B 0,C 180,E1 -14290.229,E2 -14290.229} C_VEL
LIN {X 0,Y 346.358,Z 288.886,A -85,B 0,C 180,E1 -14291.363,E2 -14291.363} C_VEL
LIN {X 0,Y 346.504,Z 283.129,A -85,B 0,C 180,E1 -14291.831,E2 -14291.831} C_VEL
LIN {X 0,Y 344.014,Z 271.204,A -85,B 0,C 180,E1 -14292.77,E2 -14292.77} C_VEL
LIN {X 0,Y 340.914,Z 258.978,A -85,B 0,C 180,E1 -14293.535,E2 -14293.535} C_VEL
LIN {X 0,Y 339.7,Z 254.444,A -85,B 0,C 180,E1 -14293.783,E2 -14293.783} C_VEL
LIN {X 0,Y 339.858,Z 251.579,A -85,B 0,C 180,E1 -14296.853,E2 -14296.853} C_VEL
LIN {X 0,Y 340.015,Z 248.278,A -85,B 0,C 180,E1 -14300.483,E2 -14300.483} C_VEL
LIN {X 0,Y 340.208,Z 246.139,A -85,B 0,C 180,E1 -14302.881,E2 -14302.881} C_VEL
LIN {X 0,Y 340.484,Z 246.074,A -85,B 0,C 180,E1 -14305.265,E2 -14305.265} C_VEL
LIN {X 0,Y 341.057,Z 246,A -85,B 0,C 180,E1 -14308.82,E2 -14308.82} C_VEL
LIN {X 0,Y 341.255,Z 245.975,A -85,B 0,C 180,E1 -14310.001,E2 -14310.001} C_VEL
LIN {X 0,Y 341.157,Z 245.986,A -85,B 0,C 180,E1 -14312.362,E2 -14312.362} C_VEL
LIN {X 0,Y 341.062,Z 246.003,A -85,B 0,C 180,E1 -14317.103,E2 -14317.103} C_VEL
LIN {X 0,Y 340.863,Z 246.024,A -85,B 0,C 180,E1 -14320.695,E2 -14320.695} C_VEL
LIN {X 0,Y 340.851,Z 246.024,A -85,B 0,C 180,E1 -14324.327,E2 -14324.327} C_VEL
LIN {X 0,Y 340.827,Z 246.028,A -85,B 0,C 180,E1 -14328.469,E2 -14328.469} C_VEL
LIN {X 0,Y 340.743,Z 246.038,A -85,B 0,C 180,E1 -14331.859,E2 -14331.859} C_VEL
LIN {X 0,Y 340.765,Z 246.035,A -85,B 0,C 180,E1 -14335.666,E2 -14335.666} C_VEL
LIN {X 0,Y 340.731,Z 246.04,A -85,B 0,C 180,E1 -14338.322,E2 -14338.322} C_VEL
LIN {X 0,Y 340.694,Z 246.047,A -85,B 0,C 180,E1 -14341.046,E2 -14341.046} C_VEL
LIN {X 0,Y 340.71,Z 246.043,A -85,B 0,C 180,E1 -14345.281,E2 -14345.281} C_VEL
LIN {X 0,Y 340.711,Z 246.045,A -85,B 0,C 180,E1 -14348.39,E2 -14348.39} C_VEL
LIN {X 0,Y 340.719,Z 246.041,A -85,B 0,C 180,E1 -14351.306,E2 -14351.306} C_VEL
LIN {X 0,Y 340.716,Z 246.044,A -85,B 0,C 180,E1 -14354.831,E2 -14354.831} C_VEL
LIN {X 0,Y 340.729,Z 246.041,A -85,B 0,C 180,E1 -14357.951,E2 -14357.951} C_VEL
LIN {X 0,Y 340.703,Z 246.044,A -85,B 0,C 180,E1 -14359.97,E2 -14359.97} C_VEL
LIN {X 0,Y 340.031,Z 246.132,A -85,B 0,C 180,E1 -14360.957,E2 -14360.957} C_VEL
LIN {X 0,Y 337.15,Z 246.49,A -85,B 0,C 180,E1 -14362.563,E2 -14362.563} C_VEL
LIN {X 0,Y 334.736,Z 246.787,A -85,B 0,C 180,E1 -14363.863,E2 -14363.863} C_VEL
LIN {X 0,Y 333.741,Z 246.911,A -85,B 0,C 180,E1 -14364.87,E2 -14364.87} C_VEL
LIN {X 0,Y 333.682,Z 246.917,A -85,B 0,C 180,E1 -14365.211,E2 -14365.211} C_VEL
LIN {X 0,Y 333.63,Z 246.928,A -85,B 0,C 180,E1 -14368.225,E2 -14368.225} C_VEL
LIN {X 0,Y 333.69,Z 246.916,A -85,B 0,C 180,E1 -14371.028,E2 -14371.028} C_VEL
LIN {X 0,Y 333.735,Z 246.912,A -85,B 0,C 180,E1 -14373.756,E2 -14373.756} C_VEL
LIN {X 0,Y 333.721,Z 246.916,A -85,B 0,C 180,E1 -14377.916,E2 -14377.916} C_VEL
LIN {X 0,Y 333.797,Z 246.904,A -85,B 0,C 180,E1 -14381.592,E2 -14381.592} C_VEL
LIN {X 0,Y 333.812,Z 246.903,A -85,B 0,C 180,E1 -14385.579,E2 -14385.579} C_VEL
LIN {X 0,Y 333.84,Z 246.897,A -85,B 0,C 180,E1 -14389.08,E2 -14389.08} C_VEL
LIN {X 0,Y 333.998,Z 246.878,A -85,B 0,C 180,E1 -14392.749,E2 -14392.749} C_VEL
LIN {X 0,Y 333.811,Z 246.901,A -85,B 0,C 180,E1 -14395.171,E2 -14395.171} C_VEL
LIN {X 0,Y 334.111,Z 246.867,A -85,B 0,C 180,E1 -14397.591,E2 -14397.591} C_VEL
LIN {X 0,Y 334.234,Z 246.852,A -85,B 0,C 180,E1 -14400.002,E2 -14400.002} C_VEL
LIN {X 0,Y 334.109,Z 246.864,A -85,B 0,C 180,E1 -14402.413,E2 -14402.413} C_VEL
LIN {X 0,Y 334.015,Z 246.878,A -85,B 0,C 180,E1 -14406.041,E2 -14406.041} C_VEL
LIN {X 0,Y 333.829,Z 246.904,A -85,B 0,C 180,E1 -14409.698,E2 -14409.698} C_VEL
LIN {X 0,Y 333.806,Z 246.906,A -85,B 0,C 180,E1 -14413.393,E2 -14413.393} C_VEL
LIN {X 0,Y 333.756,Z 246.911,A -85,B 0,C 180,E1 -14417.147,E2 -14417.147} C_VEL
LIN {X 0,Y 333.744,Z 246.912,A -85,B 0,C 180,E1 -14419.692,E2 -14419.692} C_VEL
LIN {X 0,Y 333.702,Z 246.914,A -85,B 0,C 180,E1 -14422.279,E2 -14422.279} C_VEL
LIN {X 0,Y 333.745,Z 246.909,A -85,B 0,C 180,E1 -14426.247,E2 -14426.247} C_VEL
LIN {X 0,Y 333.7,Z 246.918,A -85,B 0,C 180,E1 -14428.975,E2 -14428.975} C_VEL
LIN {X 0,Y 333.654,Z 246.921,A -85,B 0,C 180,E1 -14432.588,E2 -14432.588} C_VEL
LIN {X 0,Y 333.686,Z 246.916,A -85,B 0,C 180,E1 -14436.139,E2 -14436.139} C_VEL
LIN {X 0,Y 333.656,Z 246.925,A -85,B 0,C 180,E1 -14439.193,E2 -14439.193} C_VEL
LIN {X 0,Y 333.642,Z 246.927,A -85,B 0,C 180,E1 -14442.5,E2 -14442.5} C_VEL
LIN {X 0,Y 333.686,Z 247.146,A -85,B 0,C 180,E1 -14444.032,E2 -14444.032} C_VEL
LIN {X 0,Y 334.732,Z 252.5,A -85,B 0,C 180,E1 -14447.787,E2 -14447.787} C_VEL
LIN {X 0,Y 335.521,Z 257.476,A -85,B 0,C 180,E1 -14451.067,E2 -14451.067} C_VEL
LIN {X 0,Y 335.948,Z 261.207,A -85,B 0,C 180,E1 -14453.412,E2 -14453.412} C_VEL
LIN {X 0,Y 335.597,Z 264.864,A -85,B 0,C 180,E1 -14455.567,E2 -14455.567} C_VEL
LIN {X 0,Y 334.902,Z 269.725,A -85,B 0,C 180,E1 -14458.355,E2 -14458.355} C_VEL
LIN {X 0,Y 333.98,Z 277.017,A -85,B 0,C 180,E1 -14462.421,E2 -14462.421} C_VEL
LIN {X 0,Y 333.265,Z 284.289,A -85,B 0,C 180,E1 -14466.378,E2 -14466.378} C_VEL
LIN {X 0,Y 332.908,Z 288.832,A -85,B 0,C 180,E1 -14468.802,E2 -14468.802} C_VEL
LIN {X 0,Y 335.209,Z 302.844,A -85,B 0,C 180,E1 -14469.493,E2 -14469.493} C_VEL
LIN {X 0,Y 336.876,Z 315.529,A -85,B 0,C 180,E1 -14470.342,E2 -14470.342} C_VEL
LIN {X 0,Y 337.884,Z 327.485,A -85,B 0,C 180,E1 -14471.348,E2 -14471.348} C_VEL
LIN {X 0,Y 337.919,Z 332.406,A -85,B 0,C 180,E1 -14471.821,E2 -14471.821} C_VEL
LIN {X 0,Y 336.64,Z 343.382,A -85,B 0,C 180,E1 -14473.005,E2 -14473.005} C_VEL
LIN {X 0,Y 335.527,Z 353.499,A -85,B 0,C 180,E1 -14474.381,E2 -14474.381} C_VEL
LIN {X 0,Y 334.45,Z 363.19,A -85,B 0,C 180,E1 -14476.014,E2 -14476.014} C_VEL
LIN {X 0,Y 333.515,Z 371.862,A -85,B 0,C 180,E1 -14477.834,E2 -14477.834} C_VEL
LIN {X 0,Y 332.787,Z 378.783,A -85,B 0,C 180,E1 -14479.658,E2 -14479.658} C_VEL
LIN {X 0,Y 332.354,Z 384.324,A -85,B 0,C 180,E1 -14481.486,E2 -14481.486} C_VEL
LIN {X 0,Y 332.164,Z 388.656,A -85,B 0,C 180,E1 -14483.316,E2 -14483.316} C_VEL
LIN {X 0,Y 332.087,Z 391.893,A -85,B 0,C 180,E1 -14485.143,E2 -14485.143} C_VEL
LIN {X 0,Y 332.071,Z 393.492,A -85,B 0,C 180,E1 -14486.358,E2 -14486.358} C_VEL
LIN {X 0,Y 332.086,Z 394.675,A -85,B 0,C 180,E1 -14487.573,E2 -14487.573} C_VEL
LIN {X 0,Y 332.207,Z 395.41,A -85,B 0,C 180,E1 -14488.787,E2 -14488.787} C_VEL
LIN {X 0,Y 332.249,Z 395.734,A -85,B 0,C 180,E1 -14489.999,E2 -14489.999} C_VEL
LIN {X 0,Y 332.166,Z 395.656,A -85,B 0,C 180,E1 -14491.211,E2 -14491.211} C_VEL
LIN {X 0,Y 332.057,Z 395.181,A -85,B 0,C 180,E1 -14492.425,E2 -14492.425} C_VEL
LIN {X 0,Y 332.049,Z 394.27,A -85,B 0,C 180,E1 -14493.639,E2 -14493.639} C_VEL
LIN {X 0,Y 332.047,Z 391.568,A -85,B 0,C 180,E1 -14495.843,E2 -14495.843} C_VEL
LIN {X 0,Y 332.271,Z 387.765,A -85,B 0,C 180,E1 -14497.901,E2 -14497.901} C_VEL
LIN {X 0,Y 332.645,Z 383.242,A -85,B 0,C 180,E1 -14499.73,E2 -14499.73} C_VEL
LIN {X 0,Y 333.257,Z 377.53,A -85,B 0,C 180,E1 -14501.556,E2 -14501.556} C_VEL
LIN {X 0,Y 334.321,Z 370.449,A -85,B 0,C 180,E1 -14503.369,E2 -14503.369} C_VEL
LIN {X 0,Y 335.419,Z 362.263,A -85,B 0,C 180,E1 -14505.064,E2 -14505.064} C_VEL
LIN {X 0,Y 336.661,Z 352.679,A -85,B 0,C 180,E1 -14506.679,E2 -14506.679} C_VEL
LIN {X 0,Y 338.249,Z 341.703,A -85,B 0,C 180,E1 -14508.158,E2 -14508.158} C_VEL
LIN {X 0,Y 339.48,Z 332.246,A -85,B 0,C 180,E1 -14509.185,E2 -14509.185} C_VEL
LIN {X 0,Y 339.126,Z 321.518,A -85,B 0,C 180,E1 -14510.231,E2 -14510.231} C_VEL
LIN {X 0,Y 337.664,Z 308.727,A -85,B 0,C 180,E1 -14511.284,E2 -14511.284} C_VEL
LIN {X 0,Y 335.524,Z 297.026,A -85,B 0,C 180,E1 -14512.096,E2 -14512.096} C_VEL
LIN {X 0,Y 333.181,Z 286.848,A -85,B 0,C 180,E1 -14512.717,E2 -14512.717} C_VEL
LIN {X 0,Y 333.809,Z 280.421,A -85,B 0,C 180,E1 -14516.239,E2 -14516.239} C_VEL
LIN {X 0,Y 334.656,Z 273.37,A -85,B 0,C 180,E1 -14520.265,E2 -14520.265} C_VEL
LIN {X 0,Y 335.58,Z 267.628,A -85,B 0,C 180,E1 -14523.707,E2 -14523.707} C_VEL
LIN {X 0,Y 336.216,Z 263.106,A -85,B 0,C 180,E1 -14526.564,E2 -14526.564} C_VEL
LIN {X 0,Y 335.96,Z 259.744,A -85,B 0,C 180,E1 -14528.87,E2 -14528.87} C_VEL
LIN {X 0,Y 335.186,Z 255.425,A -85,B 0,C 180,E1 -14532.139,E2 -14532.139} C_VEL
LIN {X 0,Y 334.328,Z 250.759,A -85,B 0,C 180,E1 -14536.074,E2 -14536.074} C_VEL
LIN {X 0,Y 333.643,Z 246.928,A -85,B 0,C 180,E1 -14539.86,E2 -14539.86} C_VEL
LIN {X 0,Y 333.675,Z 246.924,A -85,B 0,C 180,E1 -14543.859,E2 -14543.859} C_VEL
LIN {X 0,Y 333.642,Z 246.927,A -85,B 0,C 180,E1 -14547.411,E2 -14547.411} C_VEL
LIN {X 0,Y 333.708,Z 246.918,A -85,B 0,C 180,E1 -14551.026,E2 -14551.026} C_VEL
LIN {X 0,Y 333.733,Z 246.916,A -85,B 0,C 180,E1 -14553.752,E2 -14553.752} C_VEL
LIN {X 0,Y 333.716,Z 246.918,A -85,B 0,C 180,E1 -14557.912,E2 -14557.912} C_VEL
LIN {X 0,Y 333.791,Z 246.907,A -85,B 0,C 180,E1 -14561.588,E2 -14561.588} C_VEL
LIN {X 0,Y 333.804,Z 246.906,A -85,B 0,C 180,E1 -14565.575,E2 -14565.575} C_VEL
LIN {X 0,Y 333.833,Z 246.902,A -85,B 0,C 180,E1 -14569.076,E2 -14569.076} C_VEL
LIN {X 0,Y 334.02,Z 246.88,A -85,B 0,C 180,E1 -14572.746,E2 -14572.746} C_VEL
LIN {X 0,Y 333.808,Z 246.907,A -85,B 0,C 180,E1 -14575.167,E2 -14575.167} C_VEL
LIN {X 0,Y 334.102,Z 246.87,A -85,B 0,C 180,E1 -14577.587,E2 -14577.587} C_VEL
LIN {X 0,Y 334.26,Z 246.85,A -85,B 0,C 180,E1 -14579.998,E2 -14579.998} C_VEL
LIN {X 0,Y 334.101,Z 246.869,A -85,B 0,C 180,E1 -14582.409,E2 -14582.409} C_VEL
LIN {X 0,Y 334.018,Z 246.878,A -85,B 0,C 180,E1 -14587.251,E2 -14587.251} C_VEL
LIN {X 0,Y 333.83,Z 246.903,A -85,B 0,C 180,E1 -14590.92,E2 -14590.92} C_VEL
LIN {X 0,Y 333.795,Z 246.912,A -85,B 0,C 180,E1 -14594.633,E2 -14594.633} C_VEL
LIN {X 0,Y 333.623,Z 246.935,A -85,B 0,C 180,E1 -14597.151,E2 -14597.151} C_VEL
LIN {X 0,Y 333.592,Z 248.594,A -85,B 0,C 180,E1 -14599.697,E2 -14599.697} C_VEL
LIN {X 0,Y 333.475,Z 250.479,A -85,B 0,C 180,E1 -14602.291,E2 -14602.291} C_VEL
LIN {X 0,Y 333.198,Z 253.542,A -85,B 0,C 180,E1 -14606.289,E2 -14606.289} C_VEL
LIN {X 0,Y 332.998,Z 256.798,A -85,B 0,C 180,E1 -14610.398,E2 -14610.398} C_VEL
LIN {X 0,Y 337.819,Z 271.104,A -85,B 0,C 180,E1 -14611.511,E2 -14611.511} C_VEL
LIN {X 0,Y 340.936,Z 283.016,A -85,B 0,C 180,E1 -14612.581,E2 -14612.581} C_VEL
LIN {X 0,Y 342.027,Z 288.895,A -85,B 0,C 180,E1 -14613.165,E2 -14613.165} C_VEL
LIN {X 0,Y 340.793,Z 300.189,A -85,B 0,C 180,E1 -14614.228,E2 -14614.228} C_VEL
LIN {X 0,Y 339.385,Z 311.46,A -85,B 0,C 180,E1 -14615.573,E2 -14615.573} C_VEL
LIN {X 0,Y 338.024,Z 321.418,A -85,B 0,C 180,E1 -14617.079,E2 -14617.079} C_VEL
LIN {X 0,Y 336.636,Z 330.464,A -85,B 0,C 180,E1 -14618.776,E2 -14618.776} C_VEL
LIN {X 0,Y 335.42,Z 337.9,A -85,B 0,C 180,E1 -14620.504,E2 -14620.504} C_VEL
LIN {X 0,Y 334.491,Z 343.907,A -85,B 0,C 180,E1 -14622.246,E2 -14622.246} C_VEL
LIN {X 0,Y 333.59,Z 349.326,A -85,B 0,C 180,E1 -14624.252,E2 -14624.252} C_VEL
LIN {X 0,Y 333.073,Z 352.727,A -85,B 0,C 180,E1 -14625.87,E2 -14625.87} C_VEL
LIN {X 0,Y 332.56,Z 355.58,A -85,B 0,C 180,E1 -14627.698,E2 -14627.698} C_VEL
LIN {X 0,Y 332.193,Z 357.524,A -85,B 0,C 180,E1 -14629.604,E2 -14629.604} C_VEL
LIN {X 0,Y 331.993,Z 358.482,A -85,B 0,C 180,E1 -14631.556,E2 -14631.556} C_VEL
LIN {X 0,Y 331.963,Z 358.363,A -85,B 0,C 180,E1 -14633.646,E2 -14633.646} C_VEL
LIN {X 0,Y 332.059,Z 357.166,A -85,B 0,C 180,E1 -14635.628,E2 -14635.628} C_VEL
LIN {X 0,Y 332.383,Z 354.666,A -85,B 0,C 180,E1 -14637.75,E2 -14637.75} C_VEL
LIN {X 0,Y 332.826,Z 350.665,A -85,B 0,C 180,E1 -14639.965,E2 -14639.965} C_VEL
LIN {X 0,Y 333.231,Z 346.498,A -85,B 0,C 180,E1 -14641.668,E2 -14641.668} C_VEL
LIN {X 0,Y 333.895,Z 341.058,A -85,B 0,C 180,E1 -14643.432,E2 -14643.432} C_VEL
LIN {X 0,Y 334.725,Z 334.399,A -85,B 0,C 180,E1 -14645.171,E2 -14645.171} C_VEL
LIN {X 0,Y 335.651,Z 326.457,A -85,B 0,C 180,E1 -14646.852,E2 -14646.852} C_VEL
LIN {X 0,Y 336.779,Z 317.277,A -85,B 0,C 180,E1 -14648.421,E2 -14648.421} C_VEL
LIN {X 0,Y 338.032,Z 306.265,A -85,B 0,C 180,E1 -14649.939,E2 -14649.939} C_VEL
LIN {X 0,Y 339.023,Z 295.664,A -85,B 0,C 180,E1 -14651.102,E2 -14651.102} C_VEL
LIN {X 0,Y 339.702,Z 284.586,A -85,B 0,C 180,E1 -14652.078,E2 -14652.078} C_VEL
LIN {X 0,Y 337.304,Z 272.869,A -85,B 0,C 180,E1 -14653.041,E2 -14653.041} C_VEL
LIN {X 0,Y 334.05,Z 259.957,A -85,B 0,C 180,E1 -14653.893,E2 -14653.893} C_VEL
LIN {X 0,Y 332.655,Z 254.81,A -85,B 0,C 180,E1 -14654.178,E2 -14654.178} C_VEL
LIN {X 0,Y 332.825,Z 251.488,A -85,B 0,C 180,E1 -14657.811,E2 -14657.811} C_VEL
LIN {X 0,Y 333.064,Z 248.178,A -85,B 0,C 180,E1 -14661.507,E2 -14661.507} C_VEL
LIN {X 0,Y 333.156,Z 247.103,A -85,B 0,C 180,E1 -14662.73,E2 -14662.73} C_VEL
LIN {X 0,Y 333.443,Z 246.95,A -85,B 0,C 180,E1 -14665.165,E2 -14665.165} C_VEL
LIN {X 0,Y 334.019,Z 246.876,A -85,B 0,C 180,E1 -14668.796,E2 -14668.796} C_VEL
LIN {X 0,Y 334.205,Z 246.853,A -85,B 0,C 180,E1 -14670.001,E2 -14670.001} C_VEL
LIN {X 0,Y 334.094,Z 246.866,A -85,B 0,C 180,E1 -14672.412,E2 -14672.412} C_VEL
LIN {X 0,Y 334.012,Z 246.882,A -85,B 0,C 180,E1 -14677.254,E2 -14677.254} C_VEL
LIN {X 0,Y 333.826,Z 246.903,A -85,B 0,C 180,E1 -14680.923,E2 -14680.923} C_VEL
LIN {X 0,Y 333.796,Z 246.904,A -85,B 0,C 180,E1 -14684.636,E2 -14684.636} C_VEL
LIN {X 0,Y 333.787,Z 246.906,A -85,B 0,C 180,E1 -14688.658,E2 -14688.658} C_VEL
LIN {X 0,Y 333.684,Z 246.917,A -85,B 0,C 180,E1 -14692.28,E2 -14692.28} C_VEL
LIN {X 0,Y 333.726,Z 246.912,A -85,B 0,C 180,E1 -14696.248,E2 -14696.248} C_VEL
LIN {X 0,Y 333.701,Z 246.919,A -85,B 0,C 180,E1 -14698.974,E2 -14698.974} C_VEL
LIN {X 0,Y 333.635,Z 246.927,A -85,B 0,C 180,E1 -14702.589,E2 -14702.589} C_VEL
LIN {X 0,Y 333.669,Z 246.92,A -85,B 0,C 180,E1 -14706.141,E2 -14706.141} C_VEL
LIN {X 0,Y 333.677,Z 246.919,A -85,B 0,C 180,E1 -14709.189,E2 -14709.189} C_VEL
LIN {X 0,Y 333.683,Z 246.922,A -85,B 0,C 180,E1 -14712.513,E2 -14712.513} C_VEL
LIN {X 0,Y 333.654,Z 246.921,A -85,B 0,C 180,E1 -14715.968,E2 -14715.968} C_VEL
LIN {X 0,Y 333.652,Z 246.921,A -85,B 0,C 180,E1 -14719.316,E2 -14719.316} C_VEL
LIN {X 0,Y 333.655,Z 246.925,A -85,B 0,C 180,E1 -14722.352,E2 -14722.352} C_VEL
LIN {X 0,Y 333.682,Z 246.917,A -85,B 0,C 180,E1 -14725.211,E2 -14725.211} C_VEL
LIN {X 0,Y 333.076,Z 246.999,A -85,B 0,C 180,E1 -14726.217,E2 -14726.217} C_VEL
LIN {X 0,Y 330.25,Z 247.358,A -85,B 0,C 180,E1 -14727.855,E2 -14727.855} C_VEL
LIN {X 0,Y 327.804,Z 247.661,A -85,B 0,C 180,E1 -14729.181,E2 -14729.181} C_VEL
LIN {X 0,Y 326.732,Z 247.789,A -85,B 0,C 180,E1 -14730.208,E2 -14730.208} C_VEL
LIN {X 0,Y 326.635,Z 247.798,A -85,B 0,C 180,E1 -14730.556,E2 -14730.556} C_VEL
LIN {X 0,Y 326.691,Z 247.791,A -85,B 0,C 180,E1 -14734.519,E2 -14734.519} C_VEL
LIN {X 0,Y 326.648,Z 247.795,A -85,B 0,C 180,E1 -14738.548,E2 -14738.548} C_VEL
LIN {X 0,Y 326.747,Z 247.78,A -85,B 0,C 180,E1 -14741.18,E2 -14741.18} C_VEL
LIN {X 0,Y 326.767,Z 247.779,A -85,B 0,C 180,E1 -14745.435,E2 -14745.435} C_VEL
LIN {X 0,Y 326.777,Z 247.777,A -85,B 0,C 180,E1 -14748.841,E2 -14748.841} C_VEL
LIN {X 0,Y 326.948,Z 247.756,A -85,B 0,C 180,E1 -14752.592,E2 -14752.592} C_VEL
LIN {X 0,Y 326.988,Z 247.756,A -85,B 0,C 180,E1 -14753.833,E2 -14753.833} C_VEL
LIN {X 0,Y 327.051,Z 247.746,A -85,B 0,C 180,E1 -14757.539,E2 -14757.539} C_VEL
LIN {X 0,Y 327.186,Z 247.73,A -85,B 0,C 180,E1 -14760.002,E2 -14760.002} C_VEL
LIN {X 0,Y 327.05,Z 247.743,A -85,B 0,C 180,E1 -14762.465,E2 -14762.465} C_VEL
LIN {X 0,Y 326.97,Z 247.754,A -85,B 0,C 180,E1 -14766.171,E2 -14766.171} C_VEL
LIN {X 0,Y 326.792,Z 247.778,A -85,B 0,C 180,E1 -14769.909,E2 -14769.909} C_VEL
LIN {X 0,Y 326.768,Z 247.782,A -85,B 0,C 180,E1 -14773.687,E2 -14773.687} C_VEL
LIN {X 0,Y 326.709,Z 247.79,A -85,B 0,C 180,E1 -14777.529,E2 -14777.529} C_VEL
LIN {X 0,Y 326.671,Z 247.791,A -85,B 0,C 180,E1 -14780.136,E2 -14780.136} C_VEL
LIN {X 0,Y 326.661,Z 247.792,A -85,B 0,C 180,E1 -14784.13,E2 -14784.13} C_VEL
LIN {X 0,Y 326.693,Z 247.789,A -85,B 0,C 180,E1 -14786.859,E2 -14786.859} C_VEL
LIN {X 0,Y 326.644,Z 247.795,A -85,B 0,C 180,E1 -14790.61,E2 -14790.61} C_VEL
LIN {X 0,Y 326.617,Z 247.797,A -85,B 0,C 180,E1 -14794.02,E2 -14794.02} C_VEL
LIN {X 0,Y 326.637,Z 247.799,A -85,B 0,C 180,E1 -14797.239,E2 -14797.239} C_VEL
LIN {X 0,Y 326.588,Z 247.806,A -85,B 0,C 180,E1 -14801.132,E2 -14801.132} C_VEL
LIN {X 0,Y 326.638,Z 247.901,A -85,B 0,C 180,E1 -14803.621,E2 -14803.621} C_VEL
LIN {X 0,Y 327.704,Z 253.471,A -85,B 0,C 180,E1 -14807.618,E2 -14807.618} C_VEL
LIN {X 0,Y 328.67,Z 259.503,A -85,B 0,C 180,E1 -14811.674,E2 -14811.674} C_VEL
LIN {X 0,Y 328.922,Z 261.987,A -85,B 0,C 180,E1 -14813.252,E2 -14813.252} C_VEL
LIN {X 0,Y 328.573,Z 265.651,A -85,B 0,C 180,E1 -14815.47,E2 -14815.47} C_VEL
LIN {X 0,Y 327.621,Z 271.858,A -85,B 0,C 180,E1 -14819.102,E2 -14819.102} C_VEL
LIN {X 0,Y 326.914,Z 277.783,A -85,B 0,C 180,E1 -14822.469,E2 -14822.469} C_VEL
LIN {X 0,Y 326.282,Z 283.817,A -85,B 0,C 180,E1 -14825.841,E2 -14825.841} C_VEL
LIN {X 0,Y 325.912,Z 288.437,A -85,B 0,C 180,E1 -14828.374,E2 -14828.374} C_VEL
LIN {X 0,Y 328.354,Z 303.589,A -85,B 0,C 180,E1 -14829.171,E2 -14829.171} C_VEL
LIN {X 0,Y 329.995,Z 316.491,A -85,B 0,C 180,E1 -14830.076,E2 -14830.076} C_VEL
LIN {X 0,Y 330.948,Z 328.192,A -85,B 0,C 180,E1 -14831.105,E2 -14831.105} C_VEL
LIN {X 0,Y 330.983,Z 332.983,A -85,B 0,C 180,E1 -14831.587,E2 -14831.587} C_VEL
LIN {X 0,Y 329.665,Z 343.72,A -85,B 0,C 180,E1 -14832.794,E2 -14832.794} C_VEL
LIN {X 0,Y 328.564,Z 353.227,A -85,B 0,C 180,E1 -14834.123,E2 -14834.123} C_VEL
LIN {X 0,Y 327.542,Z 362.485,A -85,B 0,C 180,E1 -14835.713,E2 -14835.713} C_VEL
LIN {X 0,Y 326.507,Z 371.225,A -85,B 0,C 180,E1 -14837.569,E2 -14837.569} C_VEL
LIN {X 0,Y 325.753,Z 378.193,A -85,B 0,C 180,E1 -14839.432,E2 -14839.432} C_VEL
LIN {X 0,Y 325.306,Z 383.774,A -85,B 0,C 180,E1 -14841.301,E2 -14841.301} C_VEL
LIN {X 0,Y 325.078,Z 388.141,A -85,B 0,C 180,E1 -14843.17,E2 -14843.17} C_VEL
LIN {X 0,Y 324.99,Z 391.411,A -85,B 0,C 180,E1 -14845.036,E2 -14845.036} C_VEL
LIN {X 0,Y 324.996,Z 393.026,A -85,B 0,C 180,E1 -14846.279,E2 -14846.279} C_VEL
LIN {X 0,Y 324.995,Z 394.227,A -85,B 0,C 180,E1 -14847.52,E2 -14847.52} C_VEL
LIN {X 0,Y 325.111,Z 394.987,A -85,B 0,C 180,E1 -14848.76,E2 -14848.76} C_VEL
LIN {X 0,Y 325.172,Z 395.326,A -85,B 0,C 180,E1 -14849.999,E2 -14849.999} C_VEL
LIN {X 0,Y 325.071,Z 395.26,A -85,B 0,C 180,E1 -14851.238,E2 -14851.238} C_VEL
LIN {X 0,Y 324.968,Z 394.801,A -85,B 0,C 180,E1 -14852.478,E2 -14852.478} C_VEL
LIN {X 0,Y 324.972,Z 393.915,A -85,B 0,C 180,E1 -14853.719,E2 -14853.719} C_VEL
LIN {X 0,Y 325.001,Z 390.883,A -85,B 0,C 180,E1 -14856.206,E2 -14856.206} C_VEL
LIN {X 0,Y 325.202,Z 387.463,A -85,B 0,C 180,E1 -14858.074,E2 -14858.074} C_VEL
LIN {X 0,Y 325.595,Z 382.98,A -85,B 0,C 180,E1 -14859.942,E2 -14859.942} C_VEL
LIN {X 0,Y 326.271,Z 377.317,A -85,B 0,C 180,E1 -14861.807,E2 -14861.807} C_VEL
LIN {X 0,Y 327.389,Z 370.298,A -85,B 0,C 180,E1 -14863.657,E2 -14863.657} C_VEL
LIN {X 0,Y 328.505,Z 362.493,A -85,B 0,C 180,E1 -14865.329,E2 -14865.329} C_VEL
LIN {X 0,Y 329.857,Z 352.663,A -85,B 0,C 180,E1 -14867.034,E2 -14867.034} C_VEL
LIN {X 0,Y 331.522,Z 341.789,A -85,B 0,C 180,E1 -14868.54,E2 -14868.54} C_VEL
LIN {X 0,Y 332.721,Z 332.432,A -85,B 0,C 180,E1 -14869.591,E2 -14869.591} C_VEL
LIN {X 0,Y 332.283,Z 320.815,A -85,B 0,C 180,E1 -14870.761,E2 -14870.761} C_VEL
LIN {X 0,Y 330.979,Z 309.281,A -85,B 0,C 180,E1 -14871.752,E2 -14871.752} C_VEL
LIN {X 0,Y 328.852,Z 297.479,A -85,B 0,C 180,E1 -14872.614,E2 -14872.614} C_VEL
LIN {X 0,Y 326.214,Z 286.403,A -85,B 0,C 180,E1 -14873.327,E2 -14873.327} C_VEL
LIN {X 0,Y 326.868,Z 280.185,A -85,B 0,C 180,E1 -14876.84,E2 -14876.84} C_VEL
LIN {X 0,Y 328.019,Z 272.02,A -85,B 0,C 180,E1 -14881.662,E2 -14881.662} C_VEL
LIN {X 0,Y 328.963,Z 266.353,A -85,B 0,C 180,E1 -14885.226,E2 -14885.226} C_VEL
LIN {X 0,Y 329.225,Z 264.104,A -85,B 0,C 180,E1 -14886.705,E2 -14886.705} C_VEL
LIN {X 0,Y 329.11,Z 261.875,A -85,B 0,C 180,E1 -14888.262,E2 -14888.262} C_VEL
LIN {X 0,Y 328.346,Z 257.532,A -85,B 0,C 180,E1 -14891.568,E2 -14891.568} C_VEL
LIN {X 0,Y 327.573,Z 253.365,A -85,B 0,C 180,E1 -14895.071,E2 -14895.071} C_VEL
LIN {X 0,Y 326.854,Z 249.395,A -85,B 0,C 180,E1 -14898.811,E2 -14898.811} C_VEL
LIN {X 0,Y 326.6,Z 247.805,A -85,B 0,C 180,E1 -14900.605,E2 -14900.605} C_VEL
LIN {X 0,Y 326.63,Z 247.801,A -85,B 0,C 180,E1 -14902.951,E2 -14902.951} C_VEL
LIN {X 0,Y 326.605,Z 247.804,A -85,B 0,C 180,E1 -14905.979,E2 -14905.979} C_VEL
LIN {X 0,Y 326.658,Z 247.798,A -85,B 0,C 180,E1 -14910.339,E2 -14910.339} C_VEL
LIN {X 0,Y 326.687,Z 247.793,A -85,B 0,C 180,E1 -14914.514,E2 -14914.514} C_VEL
LIN {X 0,Y 326.643,Z 247.797,A -85,B 0,C 180,E1 -14918.543,E2 -14918.543} C_VEL
LIN {X 0,Y 326.741,Z 247.786,A -85,B 0,C 180,E1 -14921.176,E2 -14921.176} C_VEL
LIN {X 0,Y 326.759,Z 247.783,A -85,B 0,C 180,E1 -14925.431,E2 -14925.431} C_VEL
LIN {X 0,Y 326.769,Z 247.782,A -85,B 0,C 180,E1 -14928.837,E2 -14928.837} C_VEL
LIN {X 0,Y 326.974,Z 247.758,A -85,B 0,C 180,E1 -14932.588,E2 -14932.588} C_VEL
LIN {X 0,Y 326.775,Z 247.783,A -85,B 0,C 180,E1 -14935.063,E2 -14935.063} C_VEL
LIN {X 0,Y 327.043,Z 247.749,A -85,B 0,C 180,E1 -14937.535,E2 -14937.535} C_VEL
LIN {X 0,Y 327.21,Z 247.728,A -85,B 0,C 180,E1 -14939.998,E2 -14939.998} C_VEL
LIN {X 0,Y 327.042,Z 247.749,A -85,B 0,C 180,E1 -14942.461,E2 -14942.461} C_VEL
LIN {X 0,Y 326.963,Z 247.756,A -85,B 0,C 180,E1 -14946.67,E2 -14946.67} C_VEL
LIN {X 0,Y 326.808,Z 247.778,A -85,B 0,C 180,E1 -14949.904,E2 -14949.904} C_VEL
LIN {X 0,Y 326.748,Z 247.789,A -85,B 0,C 180,E1 -14953.684,E2 -14953.684} C_VEL
LIN {X 0,Y 326.628,Z 247.806,A -85,B 0,C 180,E1 -14956.241,E2 -14956.241} C_VEL
LIN {X 0,Y 326.599,Z 248.227,A -85,B 0,C 180,E1 -14957.531,E2 -14957.531} C_VEL
LIN {X 0,Y 326.536,Z 250.017,A -85,B 0,C 180,E1 -14960.141,E2 -14960.141} C_VEL
LIN {X 0,Y 326.398,Z 251.904,A -85,B 0,C 180,E1 -14962.801,E2 -14962.801} C_VEL
LIN {X 0,Y 326.216,Z 253.964,A -85,B 0,C 180,E1 -14965.521,E2 -14965.521} C_VEL
LIN {X 0,Y 326.056,Z 256.122,A -85,B 0,C 180,E1 -14968.305,E2 -14968.305} C_VEL
LIN {X 0,Y 325.975,Z 257.292,A -85,B 0,C 180,E1 -14969.795,E2 -14969.795} C_VEL
LIN {X 0,Y 328.048,Z 263.057,A -85,B 0,C 180,E1 -14970.239,E2 -14970.239} C_VEL
LIN {X 0,Y 331.915,Z 274.851,A -85,B 0,C 180,E1 -14971.247,E2 -14971.247} C_VEL
LIN {X 0,Y 334.725,Z 286.417,A -85,B 0,C 180,E1 -14972.37,E2 -14972.37} C_VEL
LIN {X 0,Y 335.378,Z 291.072,A -85,B 0,C 180,E1 -14972.85,E2 -14972.85} C_VEL
LIN {X 0,Y 333.981,Z 302.663,A -85,B 0,C 180,E1 -14974.001,E2 -14974.001} C_VEL
LIN {X 0,Y 332.601,Z 312.941,A -85,B 0,C 180,E1 -14975.299,E2 -14975.299} C_VEL
LIN {X 0,Y 331.197,Z 322.53,A -85,B 0,C 180,E1 -14976.803,E2 -14976.803} C_VEL
LIN {X 0,Y 329.793,Z 331.313,A -85,B 0,C 180,E1 -14978.503,E2 -14978.503} C_VEL
LIN {X 0,Y 328.516,Z 338.651,A -85,B 0,C 180,E1 -14980.262,E2 -14980.262} C_VEL
LIN {X 0,Y 327.366,Z 345.508,A -85,B 0,C 180,E1 -14982.362,E2 -14982.362} C_VEL
LIN {X 0,Y 326.596,Z 349.954,A -85,B 0,C 180,E1 -14984.094,E2 -14984.094} C_VEL
LIN {X 0,Y 325.841,Z 354.314,A -85,B 0,C 180,E1 -14986.356,E2 -14986.356} C_VEL
LIN {X 0,Y 325.422,Z 356.504,A -85,B 0,C 180,E1 -14987.974,E2 -14987.974} C_VEL
LIN {X 0,Y 325.124,Z 358.003,A -85,B 0,C 180,E1 -14989.574,E2 -14989.574} C_VEL
LIN {X 0,Y 324.941,Z 358.783,A -85,B 0,C 180,E1 -14991.156,E2 -14991.156} C_VEL
LIN {X 0,Y 324.85,Z 358.871,A -85,B 0,C 180,E1 -14993.172,E2 -14993.172} C_VEL
LIN {X 0,Y 324.937,Z 357.853,A -85,B 0,C 180,E1 -14995.27,E2 -14995.27} C_VEL
LIN {X 0,Y 325.246,Z 355.606,A -85,B 0,C 180,E1 -14997.424,E2 -14997.424} C_VEL
LIN {X 0,Y 325.672,Z 351.846,A -85,B 0,C 180,E1 -14999.673,E2 -14999.673} C_VEL
LIN {X 0,Y 326.173,Z 347.135,A -85,B 0,C 180,E1 -15001.705,E2 -15001.705} C_VEL
LIN {X 0,Y 326.985,Z 340.664,A -85,B 0,C 180,E1 -15003.836,E2 -15003.836} C_VEL
LIN {X 0,Y 327.874,Z 333.697,A -85,B 0,C 180,E1 -15005.632,E2 -15005.632} C_VEL
LIN {X 0,Y 328.894,Z 325.305,A -85,B 0,C 180,E1 -15007.38,E2 -15007.38} C_VEL
LIN {X 0,Y 330.096,Z 315.998,A -85,B 0,C 180,E1 -15008.951,E2 -15008.951} C_VEL
LIN {X 0,Y 331.23,Z 306.031,A -85,B 0,C 180,E1 -15010.317,E2 -15010.317} C_VEL
LIN {X 0,Y 332.37,Z 294.179,A -85,B 0,C 180,E1 -15011.607,E2 -15011.607} C_VEL
LIN {X 0,Y 332.909,Z 286.044,A -85,B 0,C 180,E1 -15012.335,E2 -15012.335} C_VEL
LIN {X 0,Y 330.581,Z 274.542,A -85,B 0,C 180,E1 -15013.323,E2 -15013.323} C_VEL
LIN {X 0,Y 327.429,Z 261.865,A -85,B 0,C 180,E1 -15014.199,E2 -15014.199} C_VEL
LIN {X 0,Y 325.62,Z 255.178,A -85,B 0,C 180,E1 -15014.59,E2 -15014.59} C_VEL
LIN {X 0,Y 325.759,Z 252.508,A -85,B 0,C 180,E1 -15017.542,E2 -15017.542} C_VEL
LIN {X 0,Y 325.995,Z 249.16,A -85,B 0,C 180,E1 -15021.322,E2 -15021.322} C_VEL
LIN {X 0,Y 326.118,Z 248.072,A -85,B 0,C 180,E1 -15022.572,E2 -15022.572} C_VEL
LIN {X 0,Y 326.402,Z 247.826,A -85,B 0,C 180,E1 -15025.06,E2 -15025.06} C_VEL
LIN {X 0,Y 326.98,Z 247.753,A -85,B 0,C 180,E1 -15028.77,E2 -15028.77} C_VEL
LIN {X 0,Y 327.156,Z 247.731,A -85,B 0,C 180,E1 -15030.001,E2 -15030.001} C_VEL
LIN {X 0,Y 327.035,Z 247.745,A -85,B 0,C 180,E1 -15032.465,E2 -15032.465} C_VEL
LIN {X 0,Y 326.983,Z 247.751,A -85,B 0,C 180,E1 -15036.171,E2 -15036.171} C_VEL
LIN {X 0,Y 326.901,Z 247.763,A -85,B 0,C 180,E1 -15038.657,E2 -15038.657} C_VEL
LIN {X 0,Y 326.727,Z 247.784,A -85,B 0,C 180,E1 -15042.423,E2 -15042.423} C_VEL
LIN {X 0,Y 326.742,Z 247.786,A -85,B 0,C 180,E1 -15044.959,E2 -15044.959} C_VEL
LIN {X 0,Y 326.753,Z 247.784,A -85,B 0,C 180,E1 -15048.856,E2 -15048.856} C_VEL
LIN {X 0,Y 326.614,Z 247.801,A -85,B 0,C 180,E1 -15052.789,E2 -15052.789} C_VEL
LIN {X 0,Y 326.682,Z 247.79,A -85,B 0,C 180,E1 -15055.486,E2 -15055.486} C_VEL
LIN {X 0,Y 326.651,Z 247.793,A -85,B 0,C 180,E1 -15059.661,E2 -15059.661} C_VEL
LIN {X 0,Y 326.599,Z 247.8,A -85,B 0,C 180,E1 -15064.022,E2 -15064.022} C_VEL
LIN {X 0,Y 326.622,Z 247.798,A -85,B 0,C 180,E1 -15067.241,E2 -15067.241} C_VEL
LIN {X 0,Y 326.629,Z 247.797,A -85,B 0,C 180,E1 -15070.205,E2 -15070.205} C_VEL
LIN {X 0,Y 326.616,Z 247.797,A -85,B 0,C 180,E1 -15073.518,E2 -15073.518} C_VEL
LIN {X 0,Y 326.612,Z 247.799,A -85,B 0,C 180,E1 -15077.023,E2 -15077.023} C_VEL
LIN {X 0,Y 326.641,Z 247.794,A -85,B 0,C 180,E1 -15081.397,E2 -15081.397} C_VEL
LIN {X 0,Y 326.6,Z 247.799,A -85,B 0,C 180,E1 -15085.204,E2 -15085.204} C_VEL
LIN {X 0,Y 326.588,Z 247.801,A -85,B 0,C 180,E1 -15088.907,E2 -15088.907} C_VEL
LIN {X 0,Y 326.635,Z 247.798,A -85,B 0,C 180,E1 -15090.556,E2 -15090.556} C_VEL
LIN {X 0,Y 325.943,Z 247.883,A -85,B 0,C 180,E1 -15091.586,E2 -15091.586} C_VEL
LIN {X 0,Y 323.092,Z 248.236,A -85,B 0,C 180,E1 -15093.263,E2 -15093.263} C_VEL
LIN {X 0,Y 320.687,Z 248.538,A -85,B 0,C 180,E1 -15094.621,E2 -15094.621} C_VEL
LIN {X 0,Y 319.652,Z 248.666,A -85,B 0,C 180,E1 -15095.673,E2 -15095.673} C_VEL
LIN {X 0,Y 319.565,Z 248.673,A -85,B 0,C 180,E1 -15096.029,E2 -15096.029} C_VEL
LIN {X 0,Y 319.617,Z 248.668,A -85,B 0,C 180,E1 -15099.404,E2 -15099.404} C_VEL
LIN {X 0,Y 319.662,Z 248.668,A -85,B 0,C 180,E1 -15102.076,E2 -15102.076} C_VEL
LIN {X 0,Y 319.737,Z 248.66,A -85,B 0,C 180,E1 -15106.01,E2 -15106.01} C_VEL
LIN {X 0,Y 319.758,Z 248.656,A -85,B 0,C 180,E1 -15109.875,E2 -15109.875} C_VEL
LIN {X 0,Y 319.942,Z 248.631,A -85,B 0,C 180,E1 -15113.696,E2 -15113.696} C_VEL
LIN {X 0,Y 319.995,Z 248.624,A -85,B 0,C 180,E1 -15117.484,E2 -15117.484} C_VEL
LIN {X 0,Y 320.139,Z 248.607,A -85,B 0,C 180,E1 -15120.002,E2 -15120.002} C_VEL
LIN {X 0,Y 319.993,Z 248.622,A -85,B 0,C 180,E1 -15122.519,E2 -15122.519} C_VEL
LIN {X 0,Y 319.928,Z 248.63,A -85,B 0,C 180,E1 -15126.308,E2 -15126.308} C_VEL
LIN {X 0,Y 319.744,Z 248.654,A -85,B 0,C 180,E1 -15130.129,E2 -15130.129} C_VEL
LIN {X 0,Y 319.741,Z 248.655,A -85,B 0,C 180,E1 -15133.994,E2 -15133.994} C_VEL
LIN {X 0,Y 319.668,Z 248.663,A -85,B 0,C 180,E1 -15137.928,E2 -15137.928} C_VEL
LIN {X 0,Y 319.622,Z 248.668,A -85,B 0,C 180,E1 -15140.6,E2 -15140.6} C_VEL
LIN {X 0,Y 319.58,Z 248.679,A -85,B 0,C 180,E1 -15143.32,E2 -15143.32} C_VEL
LIN {X 0,Y 319.628,Z 248.668,A -85,B 0,C 180,E1 -15146.09,E2 -15146.09} C_VEL
LIN {X 0,Y 319.59,Z 248.675,A -85,B 0,C 180,E1 -15148.935,E2 -15148.935} C_VEL
LIN {X 0,Y 319.541,Z 248.679,A -85,B 0,C 180,E1 -15151.863,E2 -15151.863} C_VEL
LIN {X 0,Y 319.59,Z 248.674,A -85,B 0,C 180,E1 -15155.543,E2 -15155.543} C_VEL
LIN {X 0,Y 319.569,Z 248.679,A -85,B 0,C 180,E1 -15159.669,E2 -15159.669} C_VEL
LIN {X 0,Y 319.595,Z 248.884,A -85,B 0,C 180,E1 -15163.362,E2 -15163.362} C_VEL
LIN {X 0,Y 320.588,Z 254.065,A -85,B 0,C 180,E1 -15167.187,E2 -15167.187} C_VEL
LIN {X 0,Y 321.423,Z 259.037,A -85,B 0,C 180,E1 -15170.646,E2 -15170.646} C_VEL
LIN {X 0,Y 321.88,Z 262.756,A -85,B 0,C 180,E1 -15173.097,E2 -15173.097} C_VEL
LIN {X 0,Y 321.562,Z 266.425,A -85,B 0,C 180,E1 -15175.37,E2 -15175.37} C_VEL
LIN {X 0,Y 320.645,Z 272.042,A -85,B 0,C 180,E1 -15178.742,E2 -15178.742} C_VEL
LIN {X 0,Y 319.817,Z 278.511,A -85,B 0,C 180,E1 -15182.516,E2 -15182.516} C_VEL
LIN {X 0,Y 319.177,Z 284.535,A -85,B 0,C 180,E1 -15185.96,E2 -15185.96} C_VEL
LIN {X 0,Y 318.854,Z 288.104,A -85,B 0,C 180,E1 -15187.97,E2 -15187.97} C_VEL
LIN {X 0,Y 321.226,Z 302.324,A -85,B 0,C 180,E1 -15188.716,E2 -15188.716} C_VEL
LIN {X 0,Y 322.871,Z 315.111,A -85,B 0,C 180,E1 -15189.617,E2 -15189.617} C_VEL
LIN {X 0,Y 323.928,Z 327.441,A -85,B 0,C 180,E1 -15190.713,E2 -15190.713} C_VEL
LIN {X 0,Y 324.048,Z 333.511,A -85,B 0,C 180,E1 -15191.342,E2 -15191.342} C_VEL
LIN {X 0,Y 322.695,Z 344.051,A -85,B 0,C 180,E1 -15192.573,E2 -15192.573} C_VEL
LIN {X 0,Y 321.472,Z 354.295,A -85,B 0,C 180,E1 -15194.069,E2 -15194.069} C_VEL
LIN {X 0,Y 320.395,Z 363.409,A -85,B 0,C 180,E1 -15195.712,E2 -15195.712} C_VEL
LIN {X 0,Y 319.384,Z 371.838,A -85,B 0,C 180,E1 -15197.61,E2 -15197.61} C_VEL
LIN {X 0,Y 318.636,Z 378.622,A -85,B 0,C 180,E1 -15199.514,E2 -15199.514} C_VEL
LIN {X 0,Y 318.152,Z 384.844,A -85,B 0,C 180,E1 -15201.743,E2 -15201.743} C_VEL
LIN {X 0,Y 317.928,Z 389.691,A -85,B 0,C 180,E1 -15204.14,E2 -15204.14} C_VEL
LIN {X 0,Y 317.922,Z 392.56,A -85,B 0,C 180,E1 -15206.196,E2 -15206.196} C_VEL
LIN {X 0,Y 317.908,Z 393.775,A -85,B 0,C 180,E1 -15207.465,E2 -15207.465} C_VEL
LIN {X 0,Y 318.016,Z 394.565,A -85,B 0,C 180,E1 -15208.732,E2 -15208.732} C_VEL
LIN {X 0,Y 318.082,Z 394.917,A -85,B 0,C 180,E1 -15209.999,E2 -15209.999} C_VEL
LIN {X 0,Y 317.975,Z 394.864,A -85,B 0,C 180,E1 -15211.265,E2 -15211.265} C_VEL
LIN {X 0,Y 317.882,Z 394.419,A -85,B 0,C 180,E1 -15212.533,E2 -15212.533} C_VEL
LIN {X 0,Y 317.897,Z 393.564,A -85,B 0,C 180,E1 -15213.802,E2 -15213.802} C_VEL
LIN {X 0,Y 317.912,Z 390.565,A -85,B 0,C 180,E1 -15216.345,E2 -15216.345} C_VEL
LIN {X 0,Y 318.155,Z 387.185,A -85,B 0,C 180,E1 -15218.254,E2 -15218.254} C_VEL
LIN {X 0,Y 318.562,Z 382.738,A -85,B 0,C 180,E1 -15220.164,E2 -15220.164} C_VEL
LIN {X 0,Y 319.454,Z 376.076,A -85,B 0,C 180,E1 -15222.385,E2 -15222.385} C_VEL
LIN {X 0,Y 320.679,Z 368.815,A -85,B 0,C 180,E1 -15224.272,E2 -15224.272} C_VEL
LIN {X 0,Y 321.983,Z 359.749,A -85,B 0,C 180,E1 -15226.175,E2 -15226.175} C_VEL
LIN {X 0,Y 323.39,Z 350.695,A -85,B 0,C 180,E1 -15227.712,E2 -15227.712} C_VEL
LIN {X 0,Y 325.015,Z 340.682,A -85,B 0,C 180,E1 -15229.089,E2 -15229.089} C_VEL
LIN {X 0,Y 325.963,Z 332.672,A -85,B 0,C 180,E1 -15230.014,E2 -15230.014} C_VEL
LIN {X 0,Y 325.621,Z 321.742,A -85,B 0,C 180,E1 -15231.169,E2 -15231.169} C_VEL
LIN {X 0,Y 324.329,Z 309.992,A -85,B 0,C 180,E1 -15232.231,E2 -15232.231} C_VEL
LIN {X 0,Y 322.211,Z 298.188,A -85,B 0,C 180,E1 -15233.139,E2 -15233.139} C_VEL
LIN {X 0,Y 319.285,Z 286.509,A -85,B 0,C 180,E1 -15233.916,E2 -15233.916} C_VEL
LIN {X 0,Y 319.244,Z 285.979,A -85,B 0,C 180,E1 -15233.943,E2 -15233.943} C_VEL
LIN {X 0,Y 319.932,Z 279.955,A -85,B 0,C 180,E1 -15237.47,E2 -15237.47} C_VEL
LIN {X 0,Y 320.986,Z 272.995,A -85,B 0,C 180,E1 -15241.699,E2 -15241.699} C_VEL
LIN {X 0,Y 321.967,Z 267.351,A -85,B 0,C 180,E1 -15245.34,E2 -15245.34} C_VEL
LIN {X 0,Y 322.208,Z 264.006,A -85,B 0,C 180,E1 -15247.641,E2 -15247.641} C_VEL
LIN {X 0,Y 321.526,Z 259.638,A -85,B 0,C 180,E1 -15250.975,E2 -15250.975} C_VEL
LIN {X 0,Y 320.738,Z 255.446,A -85,B 0,C 180,E1 -15254.52,E2 -15254.52} C_VEL
LIN {X 0,Y 320.004,Z 251.438,A -85,B 0,C 180,E1 -15258.305,E2 -15258.305} C_VEL
LIN {X 0,Y 319.588,Z 248.678,A -85,B 0,C 180,E1 -15261.39,E2 -15261.39} C_VEL
LIN {X 0,Y 319.559,Z 248.682,A -85,B 0,C 180,E1 -15265.121,E2 -15265.121} C_VEL
LIN {X 0,Y 319.568,Z 248.682,A -85,B 0,C 180,E1 -15269.056,E2 -15269.056} C_VEL
LIN {X 0,Y 319.606,Z 248.676,A -85,B 0,C 180,E1 -15272.496,E2 -15272.496} C_VEL
LIN {X 0,Y 319.602,Z 248.676,A -85,B 0,C 180,E1 -15275.302,E2 -15275.302} C_VEL
LIN {X 0,Y 319.594,Z 248.677,A -85,B 0,C 180,E1 -15278.046,E2 -15278.046} C_VEL
LIN {X 0,Y 319.686,Z 248.665,A -85,B 0,C 180,E1 -15280.96,E2 -15280.96} C_VEL
LIN {X 0,Y 319.727,Z 248.659,A -85,B 0,C 180,E1 -15285.274,E2 -15285.274} C_VEL
LIN {X 0,Y 319.755,Z 248.656,A -85,B 0,C 180,E1 -15289.871,E2 -15289.871} C_VEL
LIN {X 0,Y 319.928,Z 248.635,A -85,B 0,C 180,E1 -15292.424,E2 -15292.424} C_VEL
LIN {X 0,Y 319.744,Z 248.658,A -85,B 0,C 180,E1 -15294.954,E2 -15294.954} C_VEL
LIN {X 0,Y 319.986,Z 248.628,A -85,B 0,C 180,E1 -15297.48,E2 -15297.48} C_VEL
LIN {X 0,Y 320.162,Z 248.606,A -85,B 0,C 180,E1 -15299.998,E2 -15299.998} C_VEL
LIN {X 0,Y 319.985,Z 248.628,A -85,B 0,C 180,E1 -15302.516,E2 -15302.516} C_VEL
LIN {X 0,Y 319.923,Z 248.634,A -85,B 0,C 180,E1 -15306.661,E2 -15306.661} C_VEL
LIN {X 0,Y 319.752,Z 248.656,A -85,B 0,C 180,E1 -15310.125,E2 -15310.125} C_VEL
LIN {X 0,Y 319.72,Z 248.664,A -85,B 0,C 180,E1 -15313.991,E2 -15313.991} C_VEL
LIN {X 0,Y 319.582,Z 248.79,A -85,B 0,C 180,E1 -15316.61,E2 -15316.61} C_VEL
LIN {X 0,Y 319.569,Z 250.52,A -85,B 0,C 180,E1 -15319.259,E2 -15319.259} C_VEL
LIN {X 0,Y 319.427,Z 252.758,A -85,B 0,C 180,E1 -15322.474,E2 -15322.474} C_VEL
LIN {X 0,Y 319.148,Z 255.452,A -85,B 0,C 180,E1 -15326.128,E2 -15326.128} C_VEL
LIN {X 0,Y 318.963,Z 257.74,A -85,B 0,C 180,E1 -15329.129,E2 -15329.129} C_VEL
LIN {X 0,Y 319.992,Z 260.836,A -85,B 0,C 180,E1 -15329.386,E2 -15329.386} C_VEL
LIN {X 0,Y 324.167,Z 272.447,A -85,B 0,C 180,E1 -15330.405,E2 -15330.405} C_VEL
LIN {X 0,Y 327.155,Z 283.318,A -85,B 0,C 180,E1 -15331.46,E2 -15331.46} C_VEL
LIN {X 0,Y 328.823,Z 292.019,A -85,B 0,C 180,E1 -15332.4,E2 -15332.4} C_VEL
LIN {X 0,Y 327.503,Z 302.578,A -85,B 0,C 180,E1 -15333.47,E2 -15333.47} C_VEL
LIN {X 0,Y 326.099,Z 312.669,A -85,B 0,C 180,E1 -15334.749,E2 -15334.749} C_VEL
LIN {X 0,Y 324.683,Z 321.868,A -85,B 0,C 180,E1 -15336.193,E2 -15336.193} C_VEL
LIN {X 0,Y 323.19,Z 330.798,A -85,B 0,C 180,E1 -15337.924,E2 -15337.924} C_VEL
LIN {X 0,Y 321.844,Z 338.147,A -85,B 0,C 180,E1 -15339.678,E2 -15339.678} C_VEL
LIN {X 0,Y 320.598,Z 345.225,A -85,B 0,C 180,E1 -15341.814,E2 -15341.814} C_VEL
LIN {X 0,Y 319.78,Z 349.663,A -85,B 0,C 180,E1 -15343.511,E2 -15343.511} C_VEL
LIN {X 0,Y 319.112,Z 353.13,A -85,B 0,C 180,E1 -15345.192,E2 -15345.192} C_VEL
LIN {X 0,Y 318.62,Z 355.764,A -85,B 0,C 180,E1 -15346.862,E2 -15346.862} C_VEL
LIN {X 0,Y 318.197,Z 357.792,A -85,B 0,C 180,E1 -15348.669,E2 -15348.669} C_VEL
LIN {X 0,Y 317.897,Z 359.071,A -85,B 0,C 180,E1 -15350.69,E2 -15350.69} C_VEL
LIN {X 0,Y 317.765,Z 359.333,A -85,B 0,C 180,E1 -15352.765,E2 -15352.765} C_VEL
LIN {X 0,Y 317.834,Z 358.486,A -85,B 0,C 180,E1 -15354.908,E2 -15354.908} C_VEL
LIN {X 0,Y 318.087,Z 356.444,A -85,B 0,C 180,E1 -15357.092,E2 -15357.092} C_VEL
LIN {X 0,Y 318.535,Z 352.739,A -85,B 0,C 180,E1 -15359.507,E2 -15359.507} C_VEL
LIN {X 0,Y 319.098,Z 347.728,A -85,B 0,C 180,E1 -15361.756,E2 -15361.756} C_VEL
LIN {X 0,Y 319.952,Z 341.281,A -85,B 0,C 180,E1 -15363.941,E2 -15363.941} C_VEL
LIN {X 0,Y 320.862,Z 334.486,A -85,B 0,C 180,E1 -15365.751,E2 -15365.751} C_VEL
LIN {X 0,Y 321.9,Z 326.162,A -85,B 0,C 180,E1 -15367.539,E2 -15367.539} C_VEL
LIN {X 0,Y 323.208,Z 316.439,A -85,B 0,C 180,E1 -15369.223,E2 -15369.223} C_VEL
LIN {X 0,Y 324.43,Z 305.723,A -85,B 0,C 180,E1 -15370.711,E2 -15370.711} C_VEL
LIN {X 0,Y 325.581,Z 294.484,A -85,B 0,C 180,E1 -15371.949,E2 -15371.949} C_VEL
LIN {X 0,Y 326.087,Z 287.419,A -85,B 0,C 180,E1 -15372.601,E2 -15372.601} C_VEL
LIN {X 0,Y 323.849,Z 276.092,A -85,B 0,C 180,E1 -15373.615,E2 -15373.615} C_VEL
LIN {X 0,Y 320.715,Z 263.526,A -85,B 0,C 180,E1 -15374.528,E2 -15374.528} C_VEL
LIN {X 0,Y 318.554,Z 255.549,A -85,B 0,C 180,E1 -15375.018,E2 -15375.018} C_VEL
LIN {X 0,Y 318.726,Z 252.404,A -85,B 0,C 180,E1 -15378.555,E2 -15378.555} C_VEL
LIN {X 0,Y 319.043,Z 249.061,A -85,B 0,C 180,E1 -15382.406,E2 -15382.406} C_VEL
LIN {X 0,Y 319.36,Z 248.703,A -85,B 0,C 180,E1 -15384.951,E2 -15384.951} C_VEL
LIN {X 0,Y 319.94,Z 248.629,A -85,B 0,C 180,E1 -15388.743,E2 -15388.743} C_VEL
LIN {X 0,Y 320.107,Z 248.609,A -85,B 0,C 180,E1 -15390.001,E2 -15390.001} C_VEL
LIN {X 0,Y 319.979,Z 248.624,A -85,B 0,C 180,E1 -15392.519,E2 -15392.519} C_VEL
LIN {X 0,Y 319.939,Z 248.629,A -85,B 0,C 180,E1 -15396.307,E2 -15396.307} C_VEL
LIN {X 0,Y 319.83,Z 248.645,A -85,B 0,C 180,E1 -15398.85,E2 -15398.85} C_VEL
LIN {X 0,Y 319.673,Z 248.664,A -85,B 0,C 180,E1 -15402.701,E2 -15402.701} C_VEL
LIN {X 0,Y 319.687,Z 248.664,A -85,B 0,C 180,E1 -15405.297,E2 -15405.297} C_VEL
LIN {X 0,Y 319.679,Z 248.665,A -85,B 0,C 180,E1 -15409.256,E2 -15409.256} C_VEL
LIN {X 0,Y 319.564,Z 248.678,A -85,B 0,C 180,E1 -15413.321,E2 -15413.321} C_VEL
LIN {X 0,Y 319.626,Z 248.669,A -85,B 0,C 180,E1 -15416.09,E2 -15416.09} C_VEL
LIN {X 0,Y 319.58,Z 248.679,A -85,B 0,C 180,E1 -15418.936,E2 -15418.936} C_VEL
LIN {X 0,Y 319.523,Z 248.681,A -85,B 0,C 180,E1 -15421.864,E2 -15421.864} C_VEL
LIN {X 0,Y 319.572,Z 248.675,A -85,B 0,C 180,E1 -15425.545,E2 -15425.545} C_VEL
LIN {X 0,Y 319.577,Z 248.675,A -85,B 0,C 180,E1 -15428.009,E2 -15428.009} C_VEL
LIN {X 0,Y 319.59,Z 248.672,A -85,B 0,C 180,E1 -15431.614,E2 -15431.614} C_VEL
LIN {X 0,Y 319.574,Z 248.675,A -85,B 0,C 180,E1 -15435.276,E2 -15435.276} C_VEL
LIN {X 0,Y 319.543,Z 248.682,A -85,B 0,C 180,E1 -15438.717,E2 -15438.717} C_VEL
LIN {X 0,Y 319.596,Z 248.676,A -85,B 0,C 180,E1 -15442.342,E2 -15442.342} C_VEL
LIN {X 0,Y 319.558,Z 248.675,A -85,B 0,C 180,E1 -15445.126,E2 -15445.126} C_VEL
LIN {X 0,Y 319.565,Z 248.675,A -85,B 0,C 180,E1 -15449.062,E2 -15449.062} C_VEL
LIN {X 0,Y 319.606,Z 248.674,A -85,B 0,C 180,E1 -15452.501,E2 -15452.501} C_VEL
LIN {X 0,Y 319.606,Z 248.67,A -85,B 0,C 180,E1 -15455.307,E2 -15455.307} C_VEL
LIN {X 0,Y 319.565,Z 248.673,A -85,B 0,C 180,E1 -15456.029,E2 -15456.029} C_VEL
LIN {X 0,Y 318.892,Z 248.759,A -85,B 0,C 180,E1 -15457.08,E2 -15457.08} C_VEL
LIN {X 0,Y 316.062,Z 249.111,A -85,B 0,C 180,E1 -15458.793,E2 -15458.793} C_VEL
LIN {X 0,Y 313.69,Z 249.41,A -85,B 0,C 180,E1 -15460.181,E2 -15460.181} C_VEL
LIN {X 0,Y 312.704,Z 249.529,A -85,B 0,C 180,E1 -15461.255,E2 -15461.255} C_VEL
LIN {X 0,Y 312.639,Z 249.538,A -85,B 0,C 180,E1 -15461.618,E2 -15461.618} C_VEL
LIN {X 0,Y 312.698,Z 249.533,A -85,B 0,C 180,E1 -15465.689,E2 -15465.689} C_VEL
LIN {X 0,Y 312.704,Z 249.533,A -85,B 0,C 180,E1 -15469.644,E2 -15469.644} C_VEL
LIN {X 0,Y 312.898,Z 249.507,A -85,B 0,C 180,E1 -15473.554,E2 -15473.554} C_VEL
LIN {X 0,Y 312.941,Z 249.502,A -85,B 0,C 180,E1 -15477.428,E2 -15477.428} C_VEL
LIN {X 0,Y 313.092,Z 249.485,A -85,B 0,C 180,E1 -15480.002,E2 -15480.002} C_VEL
LIN {X 0,Y 312.94,Z 249.501,A -85,B 0,C 180,E1 -15482.576,E2 -15482.576} C_VEL
LIN {X 0,Y 312.871,Z 249.508,A -85,B 0,C 180,E1 -15486.451,E2 -15486.451} C_VEL
LIN {X 0,Y 312.759,Z 249.523,A -85,B 0,C 180,E1 -15489.052,E2 -15489.052} C_VEL
LIN {X 0,Y 312.643,Z 249.539,A -85,B 0,C 180,E1 -15492.993,E2 -15492.993} C_VEL
LIN {X 0,Y 312.648,Z 249.541,A -85,B 0,C 180,E1 -15495.651,E2 -15495.651} C_VEL
LIN {X 0,Y 312.639,Z 249.541,A -85,B 0,C 180,E1 -15499.237,E2 -15499.237} C_VEL
LIN {X 0,Y 312.556,Z 249.55,A -85,B 0,C 180,E1 -15502.79,E2 -15502.79} C_VEL
LIN {X 0,Y 312.607,Z 249.543,A -85,B 0,C 180,E1 -15505.934,E2 -15505.934} C_VEL
LIN {X 0,Y 312.548,Z 249.552,A -85,B 0,C 180,E1 -15509.651,E2 -15509.651} C_VEL
LIN {X 0,Y 312.53,Z 249.553,A -85,B 0,C 180,E1 -15513.689,E2 -15513.689} C_VEL
LIN {X 0,Y 312.53,Z 249.555,A -85,B 0,C 180,E1 -15517.386,E2 -15517.386} C_VEL
LIN {X 0,Y 312.5,Z 249.56,A -85,B 0,C 180,E1 -15520.709,E2 -15520.709} C_VEL
LIN {X 0,Y 312.557,Z 249.665,A -85,B 0,C 180,E1 -15522.97,E2 -15522.97} C_VEL
LIN {X 0,Y 313.466,Z 254.703,A -85,B 0,C 180,E1 -15526.775,E2 -15526.775} C_VEL
LIN {X 0,Y 314.378,Z 259.801,A -85,B 0,C 180,E1 -15530.421,E2 -15530.421} C_VEL
LIN {X 0,Y 314.835,Z 263.53,A -85,B 0,C 180,E1 -15532.934,E2 -15532.934} C_VEL
LIN {X 0,Y 314.535,Z 267.102,A -85,B 0,C 180,E1 -15535.217,E2 -15535.217} C_VEL
LIN {X 0,Y 313.515,Z 273.216,A -85,B 0,C 180,E1 -15538.962,E2 -15538.962} C_VEL
LIN {X 0,Y 312.741,Z 279.24,A -85,B 0,C 180,E1 -15542.567,E2 -15542.567} C_VEL
LIN {X 0,Y 311.951,Z 286.443,A -85,B 0,C 180,E1 -15546.779,E2 -15546.779} C_VEL
LIN {X 0,Y 311.822,Z 287.749,A -85,B 0,C 180,E1 -15547.533,E2 -15547.533} C_VEL
LIN {X 0,Y 314.176,Z 301.782,A -85,B 0,C 180,E1 -15548.288,E2 -15548.288} C_VEL
LIN {X 0,Y 315.886,Z 314.94,A -85,B 0,C 180,E1 -15549.243,E2 -15549.243} C_VEL
LIN {X 0,Y 316.888,Z 326.551,A -85,B 0,C 180,E1 -15550.301,E2 -15550.301} C_VEL
LIN {X 0,Y 317.103,Z 333.888,A -85,B 0,C 180,E1 -15551.085,E2 -15551.085} C_VEL
LIN {X 0,Y 315.729,Z 344.296,A -85,B 0,C 180,E1 -15552.344,E2 -15552.344} C_VEL
LIN {X 0,Y 314.53,Z 354.054,A -85,B 0,C 180,E1 -15553.809,E2 -15553.809} C_VEL
LIN {X 0,Y 313.496,Z 362.653,A -85,B 0,C 180,E1 -15555.391,E2 -15555.391} C_VEL
LIN {X 0,Y 312.415,Z 371.169,A -85,B 0,C 180,E1 -15557.329,E2 -15557.329} C_VEL
LIN {X 0,Y 311.608,Z 378.002,A -85,B 0,C 180,E1 -15559.275,E2 -15559.275} C_VEL
LIN {X 0,Y 311.09,Z 384.278,A -85,B 0,C 180,E1 -15561.555,E2 -15561.555} C_VEL
LIN {X 0,Y 310.898,Z 388.343,A -85,B 0,C 180,E1 -15563.509,E2 -15563.509} C_VEL
LIN {X 0,Y 310.813,Z 390.433,A -85,B 0,C 180,E1 -15564.809,E2 -15564.809} C_VEL
LIN {X 0,Y 310.849,Z 392.084,A -85,B 0,C 180,E1 -15566.11,E2 -15566.11} C_VEL
LIN {X 0,Y 310.824,Z 393.315,A -85,B 0,C 180,E1 -15567.407,E2 -15567.407} C_VEL
LIN {X 0,Y 310.921,Z 394.135,A -85,B 0,C 180,E1 -15568.703,E2 -15568.703} C_VEL
LIN {X 0,Y 310.992,Z 394.507,A -85,B 0,C 180,E1 -15569.999,E2 -15569.999} C_VEL
LIN {X 0,Y 310.88,Z 394.47,A -85,B 0,C 180,E1 -15571.294,E2 -15571.294} C_VEL
LIN {X 0,Y 310.799,Z 394.041,A -85,B 0,C 180,E1 -15572.591,E2 -15572.591} C_VEL
LIN {X 0,Y 310.8,Z 393.214,A -85,B 0,C 180,E1 -15573.888,E2 -15573.888} C_VEL
LIN {X 0,Y 310.835,Z 390.252,A -85,B 0,C 180,E1 -15576.49,E2 -15576.49} C_VEL
LIN {X 0,Y 311.094,Z 386.905,A -85,B 0,C 180,E1 -15578.443,E2 -15578.443} C_VEL
LIN {X 0,Y 311.546,Z 382.495,A -85,B 0,C 180,E1 -15580.396,E2 -15580.396} C_VEL
LIN {X 0,Y 312.504,Z 375.879,A -85,B 0,C 180,E1 -15582.665,E2 -15582.665} C_VEL
LIN {X 0,Y 313.759,Z 368.699,A -85,B 0,C 180,E1 -15584.594,E2 -15584.594} C_VEL
LIN {X 0,Y 315.237,Z 359.223,A -85,B 0,C 180,E1 -15586.632,E2 -15586.632} C_VEL
LIN {X 0,Y 316.831,Z 349.778,A -85,B 0,C 180,E1 -15588.258,E2 -15588.258} C_VEL
LIN {X 0,Y 318.541,Z 339.618,A -85,B 0,C 180,E1 -15589.66,E2 -15589.66} C_VEL
LIN {X 0,Y 319.231,Z 332.957,A -85,B 0,C 180,E1 -15590.455,E2 -15590.455} C_VEL
LIN {X 0,Y 318.943,Z 322.534,A -85,B 0,C 180,E1 -15591.601,E2 -15591.601} C_VEL
LIN {X 0,Y 317.59,Z 309.766,A -85,B 0,C 180,E1 -15592.807,E2 -15592.807} C_VEL
LIN {X 0,Y 315.192,Z 297.016,A -85,B 0,C 180,E1 -15593.835,E2 -15593.835} C_VEL
LIN {X 0,Y 312.383,Z 286.175,A -85,B 0,C 180,E1 -15594.594,E2 -15594.594} C_VEL
LIN {X 0,Y 312.33,Z 285.501,A -85,B 0,C 180,E1 -15594.642,E2 -15594.642} C_VEL
LIN {X 0,Y 312.989,Z 279.731,A -85,B 0,C 180,E1 -15598.133,E2 -15598.133} C_VEL
LIN {X 0,Y 314.181,Z 272.84,A -85,B 0,C 180,E1 -15602.469,E2 -15602.469} C_VEL
LIN {X 0,Y 314.97,Z 268.339,A -85,B 0,C 180,E1 -15605.459,E2 -15605.459} C_VEL
LIN {X 0,Y 315.211,Z 265.013,A -85,B 0,C 180,E1 -15607.815,E2 -15607.815} C_VEL
LIN {X 0,Y 314.644,Z 261.475,A -85,B 0,C 180,E1 -15610.583,E2 -15610.583} C_VEL
LIN {X 0,Y 313.841,Z 257.215,A -85,B 0,C 180,E1 -15614.224,E2 -15614.224} C_VEL
LIN {X 0,Y 313.166,Z 253.48,A -85,B 0,C 180,E1 -15617.779,E2 -15617.779} C_VEL
LIN {X 0,Y 312.711,Z 250.448,A -85,B 0,C 180,E1 -15621.001,E2 -15621.001} C_VEL
LIN {X 0,Y 312.539,Z 249.556,A -85,B 0,C 180,E1 -15622.262,E2 -15622.262} C_VEL
LIN {X 0,Y 312.518,Z 249.559,A -85,B 0,C 180,E1 -15626.309,E2 -15626.309} C_VEL
LIN {X 0,Y 312.543,Z 249.556,A -85,B 0,C 180,E1 -15630.348,E2 -15630.348} C_VEL
LIN {X 0,Y 312.6,Z 249.548,A -85,B 0,C 180,E1 -15634.062,E2 -15634.062} C_VEL
LIN {X 0,Y 312.584,Z 249.549,A -85,B 0,C 180,E1 -15637.527,E2 -15637.527} C_VEL
LIN {X 0,Y 312.635,Z 249.542,A -85,B 0,C 180,E1 -15641.654,E2 -15641.654} C_VEL
LIN {X 0,Y 312.69,Z 249.535,A -85,B 0,C 180,E1 -15645.684,E2 -15645.684} C_VEL
LIN {X 0,Y 312.699,Z 249.535,A -85,B 0,C 180,E1 -15649.64,E2 -15649.64} C_VEL
LIN {X 0,Y 312.867,Z 249.515,A -85,B 0,C 180,E1 -15652.252,E2 -15652.252} C_VEL
LIN {X 0,Y 312.714,Z 249.533,A -85,B 0,C 180,E1 -15654.84,E2 -15654.84} C_VEL
LIN {X 0,Y 312.985,Z 249.5,A -85,B 0,C 180,E1 -15658.711,E2 -15658.711} C_VEL
LIN {X 0,Y 313.113,Z 249.484,A -85,B 0,C 180,E1 -15659.998,E2 -15659.998} C_VEL
LIN {X 0,Y 312.932,Z 249.506,A -85,B 0,C 180,E1 -15662.572,E2 -15662.572} C_VEL
LIN {X 0,Y 312.886,Z 249.51,A -85,B 0,C 180,E1 -15666.644,E2 -15666.644} C_VEL
LIN {X 0,Y 312.779,Z 249.524,A -85,B 0,C 180,E1 -15669.047,E2 -15669.047} C_VEL
LIN {X 0,Y 312.627,Z 249.545,A -85,B 0,C 180,E1 -15672.989,E2 -15672.989} C_VEL
LIN {X 0,Y 312.565,Z 249.558,A -85,B 0,C 180,E1 -15675.651,E2 -15675.651} C_VEL
LIN {X 0,Y 312.563,Z 251.623,A -85,B 0,C 180,E1 -15679.205,E2 -15679.205} C_VEL
LIN {X 0,Y 312.371,Z 254.022,A -85,B 0,C 180,E1 -15682.716,E2 -15682.716} C_VEL
LIN {X 0,Y 312.072,Z 256.959,A -85,B 0,C 180,E1 -15686.767,E2 -15686.767} C_VEL
LIN {X 0,Y 312.012,Z 258.424,A -85,B 0,C 180,E1 -15688.479,E2 -15688.479} C_VEL
LIN {X 0,Y 314.007,Z 263.859,A -85,B 0,C 180,E1 -15688.927,E2 -15688.927} C_VEL
LIN {X 0,Y 317.591,Z 273.742,A -85,B 0,C 180,E1 -15689.859,E2 -15689.859} C_VEL
LIN {X 0,Y 320.614,Z 284.857,A -85,B 0,C 180,E1 -15691.004,E2 -15691.004} C_VEL
LIN {X 0,Y 322.208,Z 293.941,A -85,B 0,C 180,E1 -15692.023,E2 -15692.023} C_VEL
LIN {X 0,Y 320.683,Z 305.074,A -85,B 0,C 180,E1 -15693.22,E2 -15693.22} C_VEL
LIN {X 0,Y 319.051,Z 315.936,A -85,B 0,C 180,E1 -15694.704,E2 -15694.704} C_VEL
LIN {X 0,Y 317.561,Z 325.157,A -85,B 0,C 180,E1 -15696.272,E2 -15696.272} C_VEL
LIN {X 0,Y 316.152,Z 332.809,A -85,B 0,C 180,E1 -15697.862,E2 -15697.862} C_VEL
LIN {X 0,Y 314.806,Z 339.76,A -85,B 0,C 180,E1 -15699.631,E2 -15699.631} C_VEL
LIN {X 0,Y 313.538,Z 346.533,A -85,B 0,C 180,E1 -15701.817,E2 -15701.817} C_VEL
LIN {X 0,Y 312.518,Z 351.687,A -85,B 0,C 180,E1 -15703.978,E2 -15703.978} C_VEL
LIN {X 0,Y 311.735,Z 355.529,A -85,B 0,C 180,E1 -15706.169,E2 -15706.169} C_VEL
LIN {X 0,Y 311.222,Z 357.925,A -85,B 0,C 180,E1 -15708.173,E2 -15708.173} C_VEL
LIN {X 0,Y 310.817,Z 359.528,A -85,B 0,C 180,E1 -15710.721,E2 -15710.721} C_VEL
LIN {X 0,Y 310.682,Z 359.79,A -85,B 0,C 180,E1 -15712.356,E2 -15712.356} C_VEL
LIN {X 0,Y 310.728,Z 359.133,A -85,B 0,C 180,E1 -15714.508,E2 -15714.508} C_VEL
LIN {X 0,Y 310.968,Z 357.278,A -85,B 0,C 180,E1 -15716.738,E2 -15716.738} C_VEL
LIN {X 0,Y 311.349,Z 354.037,A -85,B 0,C 180,E1 -15719.061,E2 -15719.061} C_VEL
LIN {X 0,Y 311.811,Z 350.397,A -85,B 0,C 180,E1 -15720.921,E2 -15720.921} C_VEL
LIN {X 0,Y 312.565,Z 344.311,A -85,B 0,C 180,E1 -15723.277,E2 -15723.277} C_VEL
LIN {X 0,Y 313.435,Z 338.082,A -85,B 0,C 180,E1 -15725.14,E2 -15725.14} C_VEL
LIN {X 0,Y 314.444,Z 330.479,A -85,B 0,C 180,E1 -15726.976,E2 -15726.976} C_VEL
LIN {X 0,Y 315.763,Z 320.927,A -85,B 0,C 180,E1 -15728.833,E2 -15728.833} C_VEL
LIN {X 0,Y 317.048,Z 310.766,A -85,B 0,C 180,E1 -15730.412,E2 -15730.412} C_VEL
LIN {X 0,Y 318.339,Z 299.094,A -85,B 0,C 180,E1 -15731.853,E2 -15731.853} C_VEL
LIN {X 0,Y 319.257,Z 288.71,A -85,B 0,C 180,E1 -15732.876,E2 -15732.876} C_VEL
LIN {X 0,Y 317.175,Z 277.992,A -85,B 0,C 180,E1 -15733.886,E2 -15733.886} C_VEL
LIN {X 0,Y 314.073,Z 265.365,A -85,B 0,C 180,E1 -15734.859,E2 -15734.859} C_VEL
LIN {X 0,Y 311.557,Z 255.889,A -85,B 0,C 180,E1 -15735.484,E2 -15735.484} C_VEL
LIN {X 0,Y 311.736,Z 252.306,A -85,B 0,C 180,E1 -15739.611,E2 -15739.611} C_VEL
LIN {X 0,Y 311.983,Z 249.941,A -85,B 0,C 180,E1 -15742.365,E2 -15742.365} C_VEL
LIN {X 0,Y 312.317,Z 249.58,A -85,B 0,C 180,E1 -15744.837,E2 -15744.837} C_VEL
LIN {X 0,Y 312.899,Z 249.507,A -85,B 0,C 180,E1 -15748.714,E2 -15748.714} C_VEL
LIN {X 0,Y 312.979,Z 249.501,A -85,B 0,C 180,E1 -15751.288,E2 -15751.288} C_VEL
LIN {X 0,Y 312.706,Z 249.534,A -85,B 0,C 180,E1 -15755.159,E2 -15755.159} C_VEL
LIN {X 0,Y 312.858,Z 249.512,A -85,B 0,C 180,E1 -15757.747,E2 -15757.747} C_VEL
LIN {X 0,Y 312.66,Z 249.537,A -85,B 0,C 180,E1 -15761.673,E2 -15761.673} C_VEL
LIN {X 0,Y 312.688,Z 249.535,A -85,B 0,C 180,E1 -15764.889,E2 -15764.889} C_VEL
LIN {X 0,Y 312.634,Z 249.543,A -85,B 0,C 180,E1 -15769.246,E2 -15769.246} C_VEL
LIN {X 0,Y 312.538,Z 249.554,A -85,B 0,C 180,E1 -15772.792,E2 -15772.792} C_VEL
LIN {X 0,Y 312.573,Z 249.551,A -85,B 0,C 180,E1 -15776.725,E2 -15776.725} C_VEL
LIN {X 0,Y 312.536,Z 249.552,A -85,B 0,C 180,E1 -15779.652,E2 -15779.652} C_VEL
LIN {X 0,Y 312.511,Z 249.554,A -85,B 0,C 180,E1 -15783.691,E2 -15783.691} C_VEL
LIN {X 0,Y 312.534,Z 249.552,A -85,B 0,C 180,E1 -15787.385,E2 -15787.385} C_VEL
LIN {X 0,Y 312.519,Z 249.558,A -85,B 0,C 180,E1 -15790.706,E2 -15790.706} C_VEL
LIN {X 0,Y 312.53,Z 249.554,A -85,B 0,C 180,E1 -15794.197,E2 -15794.197} C_VEL
LIN {X 0,Y 312.529,Z 249.553,A -85,B 0,C 180,E1 -15797.911,E2 -15797.911} C_VEL
LIN {X 0,Y 312.554,Z 249.55,A -85,B 0,C 180,E1 -15801.908,E2 -15801.908} C_VEL
LIN {X 0,Y 312.504,Z 249.553,A -85,B 0,C 180,E1 -15805.793,E2 -15805.793} C_VEL
LIN {X 0,Y 312.519,Z 249.554,A -85,B 0,C 180,E1 -15808.856,E2 -15808.856} C_VEL
LIN {X 0,Y 312.57,Z 249.549,A -85,B 0,C 180,E1 -15811.827,E2 -15811.827} C_VEL
LIN {X 0,Y 312.586,Z 249.546,A -85,B 0,C 180,E1 -15814.714,E2 -15814.714} C_VEL
LIN {X 0,Y 312.589,Z 249.544,A -85,B 0,C 180,E1 -15817.532,E2 -15817.532} C_VEL
LIN {X 0,Y 312.639,Z 249.538,A -85,B 0,C 180,E1 -15821.618,E2 -15821.618} C_VEL
LIN {X 0,Y 312.009,Z 249.621,A -85,B 0,C 180,E1 -15822.695,E2 -15822.695} C_VEL
LIN {X 0,Y 309.149,Z 249.976,A -85,B 0,C 180,E1 -15824.447,E2 -15824.447} C_VEL
LIN {X 0,Y 306.704,Z 250.281,A -85,B 0,C 180,E1 -15825.867,E2 -15825.867} C_VEL
LIN {X 0,Y 305.661,Z 250.408,A -85,B 0,C 180,E1 -15826.968,E2 -15826.968} C_VEL
LIN {X 0,Y 305.581,Z 250.417,A -85,B 0,C 180,E1 -15827.341,E2 -15827.341} C_VEL
LIN {X 0,Y 305.761,Z 250.395,A -85,B 0,C 180,E1 -15831.26,E2 -15831.26} C_VEL
LIN {X 0,Y 305.838,Z 250.384,A -85,B 0,C 180,E1 -15833.404,E2 -15833.404} C_VEL
LIN {X 0,Y 305.89,Z 250.379,A -85,B 0,C 180,E1 -15837.368,E2 -15837.368} C_VEL
LIN {X 0,Y 306.046,Z 250.363,A -85,B 0,C 180,E1 -15840.002,E2 -15840.002} C_VEL
LIN {X 0,Y 305.888,Z 250.379,A -85,B 0,C 180,E1 -15842.636,E2 -15842.636} C_VEL
LIN {X 0,Y 305.816,Z 250.386,A -85,B 0,C 180,E1 -15846.6,E2 -15846.6} C_VEL
LIN {X 0,Y 305.703,Z 250.403,A -85,B 0,C 180,E1 -15849.263,E2 -15849.263} C_VEL
LIN {X 0,Y 305.598,Z 250.419,A -85,B 0,C 180,E1 -15853.298,E2 -15853.298} C_VEL
LIN {X 0,Y 305.603,Z 250.415,A -85,B 0,C 180,E1 -15856.021,E2 -15856.021} C_VEL
LIN {X 0,Y 305.586,Z 250.42,A -85,B 0,C 180,E1 -15859.446,E2 -15859.446} C_VEL
LIN {X 0,Y 305.5,Z 250.43,A -85,B 0,C 180,E1 -15863.042,E2 -15863.042} C_VEL
LIN {X 0,Y 305.536,Z 250.423,A -85,B 0,C 180,E1 -15866.22,E2 -15866.22} C_VEL
LIN {X 0,Y 305.499,Z 250.43,A -85,B 0,C 180,E1 -15869.048,E2 -15869.048} C_VEL
LIN {X 0,Y 305.452,Z 250.434,A -85,B 0,C 180,E1 -15871.953,E2 -15871.953} C_VEL
LIN {X 0,Y 305.473,Z 250.436,A -85,B 0,C 180,E1 -15875.114,E2 -15875.114} C_VEL
LIN {X 0,Y 305.45,Z 250.435,A -85,B 0,C 180,E1 -15878.527,E2 -15878.527} C_VEL
LIN {X 0,Y 305.501,Z 250.504,A -85,B 0,C 180,E1 -15882.593,E2 -15882.593} C_VEL
LIN {X 0,Y 306.581,Z 256.437,A -85,B 0,C 180,E1 -15887.188,E2 -15887.188} C_VEL
LIN {X 0,Y 307.463,Z 261.715,A -85,B 0,C 180,E1 -15891.005,E2 -15891.005} C_VEL
LIN {X 0,Y 307.774,Z 265.489,A -85,B 0,C 180,E1 -15893.578,E2 -15893.578} C_VEL
LIN {X 0,Y 307.073,Z 270.312,A -85,B 0,C 180,E1 -15896.68,E2 -15896.68} C_VEL
LIN {X 0,Y 305.971,Z 277.541,A -85,B 0,C 180,E1 -15901.159,E2 -15901.159} C_VEL
LIN {X 0,Y 305.094,Z 284.73,A -85,B 0,C 180,E1 -15905.502,E2 -15905.502} C_VEL
LIN {X 0,Y 304.806,Z 287.414,A -85,B 0,C 180,E1 -15907.085,E2 -15907.085} C_VEL
LIN {X 0,Y 307.117,Z 300.82,A -85,B 0,C 180,E1 -15907.815,E2 -15907.815} C_VEL
LIN {X 0,Y 308.812,Z 313.921,A -85,B 0,C 180,E1 -15908.781,E2 -15908.781} C_VEL
LIN {X 0,Y 309.883,Z 325.701,A -85,B 0,C 180,E1 -15909.875,E2 -15909.875} C_VEL
LIN {X 0,Y 310.161,Z 334.259,A -85,B 0,C 180,E1 -15910.817,E2 -15910.817} C_VEL
LIN {X 0,Y 308.641,Z 345.709,A -85,B 0,C 180,E1 -15912.267,E2 -15912.267} C_VEL
LIN {X 0,Y 307.327,Z 355.555,A -85,B 0,C 180,E1 -15913.839,E2 -15913.839} C_VEL
LIN {X 0,Y 306.348,Z 363.454,A -85,B 0,C 180,E1 -15915.382,E2 -15915.382} C_VEL
LIN {X 0,Y 305.28,Z 371.729,A -85,B 0,C 180,E1 -15917.366,E2 -15917.366} C_VEL
LIN {X 0,Y 304.489,Z 378.39,A -85,B 0,C 180,E1 -15919.358,E2 -15919.358} C_VEL
LIN {X 0,Y 304.019,Z 383.694,A -85,B 0,C 180,E1 -15921.357,E2 -15921.357} C_VEL
LIN {X 0,Y 303.828,Z 387.804,A -85,B 0,C 180,E1 -15923.357,E2 -15923.357} C_VEL
LIN {X 0,Y 303.724,Z 389.933,A -85,B 0,C 180,E1 -15924.688,E2 -15924.688} C_VEL
LIN {X 0,Y 303.777,Z 391.604,A -85,B 0,C 180,E1 -15926.019,E2 -15926.019} C_VEL
LIN {X 0,Y 303.826,Z 393.699,A -85,B 0,C 180,E1 -15928.673,E2 -15928.673} C_VEL
LIN {X 0,Y 303.902,Z 394.096,A -85,B 0,C 180,E1 -15929.999,E2 -15929.999} C_VEL
LIN {X 0,Y 303.785,Z 394.075,A -85,B 0,C 180,E1 -15931.324,E2 -15931.324} C_VEL
LIN {X 0,Y 303.717,Z 393.663,A -85,B 0,C 180,E1 -15932.651,E2 -15932.651} C_VEL
LIN {X 0,Y 303.707,Z 392.859,A -85,B 0,C 180,E1 -15933.979,E2 -15933.979} C_VEL
LIN {X 0,Y 303.68,Z 391.226,A -85,B 0,C 180,E1 -15935.639,E2 -15935.639} C_VEL
LIN {X 0,Y 303.925,Z 387.853,A -85,B 0,C 180,E1 -15937.974,E2 -15937.974} C_VEL
LIN {X 0,Y 304.32,Z 383.852,A -85,B 0,C 180,E1 -15939.973,E2 -15939.973} C_VEL
LIN {X 0,Y 305.002,Z 378.735,A -85,B 0,C 180,E1 -15941.968,E2 -15941.968} C_VEL
LIN {X 0,Y 306.196,Z 372.361,A -85,B 0,C 180,E1 -15943.944,E2 -15943.944} C_VEL
LIN {X 0,Y 307.577,Z 364.44,A -85,B 0,C 180,E1 -15945.913,E2 -15945.913} C_VEL
LIN {X 0,Y 309.183,Z 354.629,A -85,B 0,C 180,E1 -15947.869,E2 -15947.869} C_VEL
LIN {X 0,Y 311.01,Z 344.543,A -85,B 0,C 180,E1 -15949.468,E2 -15949.468} C_VEL
LIN {X 0,Y 312.461,Z 335.997,A -85,B 0,C 180,E1 -15950.574,E2 -15950.574} C_VEL
LIN {X 0,Y 312.386,Z 324.527,A -85,B 0,C 180,E1 -15951.927,E2 -15951.927} C_VEL
LIN {X 0,Y 311.176,Z 311.793,A -85,B 0,C 180,E1 -15953.213,E2 -15953.213} C_VEL
LIN {X 0,Y 308.969,Z 299.256,A -85,B 0,C 180,E1 -15954.305,E2 -15954.305} C_VEL
LIN {X 0,Y 305.401,Z 285.054,A -85,B 0,C 180,E1 -15955.366,E2 -15955.366} C_VEL
LIN {X 0,Y 306.181,Z 278.818,A -85,B 0,C 180,E1 -15959.277,E2 -15959.277} C_VEL
LIN {X 0,Y 307.023,Z 274.427,A -85,B 0,C 180,E1 -15962.115,E2 -15962.115} C_VEL
LIN {X 0,Y 307.98,Z 269.323,A -85,B 0,C 180,E1 -15965.583,E2 -15965.583} C_VEL
LIN {X 0,Y 308.178,Z 266.015,A -85,B 0,C 180,E1 -15968.003,E2 -15968.003} C_VEL
LIN {X 0,Y 307.439,Z 261.675,A -85,B 0,C 180,E1 -15971.522,E2 -15971.522} C_VEL
LIN {X 0,Y 306.665,Z 257.488,A -85,B 0,C 180,E1 -15975.269,E2 -15975.269} C_VEL
LIN {X 0,Y 306.021,Z 253.571,A -85,B 0,C 180,E1 -15979.275,E2 -15979.275} C_VEL
LIN {X 0,Y 305.465,Z 250.438,A -85,B 0,C 180,E1 -15982.948,E2 -15982.948} C_VEL
LIN {X 0,Y 305.464,Z 250.438,A -85,B 0,C 180,E1 -15986.481,E2 -15986.481} C_VEL
LIN {X 0,Y 305.461,Z 250.437,A -85,B 0,C 180,E1 -15989.589,E2 -15989.589} C_VEL
LIN {X 0,Y 305.519,Z 250.431,A -85,B 0,C 180,E1 -15992.606,E2 -15992.606} C_VEL
LIN {X 0,Y 305.505,Z 250.432,A -85,B 0,C 180,E1 -15995.537,E2 -15995.537} C_VEL
LIN {X 0,Y 305.516,Z 250.429,A -85,B 0,C 180,E1 -15999.813,E2 -15999.813} C_VEL
LIN {X 0,Y 305.571,Z 250.422,A -85,B 0,C 180,E1 -16002.601,E2 -16002.601} C_VEL
LIN {X 0,Y 305.645,Z 250.413,A -85,B 0,C 180,E1 -16005.347,E2 -16005.347} C_VEL
LIN {X 0,Y 305.636,Z 250.416,A -85,B 0,C 180,E1 -16009.398,E2 -16009.398} C_VEL
LIN {X 0,Y 305.808,Z 250.394,A -85,B 0,C 180,E1 -16012.072,E2 -16012.072} C_VEL
LIN {X 0,Y 305.685,Z 250.408,A -85,B 0,C 180,E1 -16014.721,E2 -16014.721} C_VEL
LIN {X 0,Y 305.951,Z 250.376,A -85,B 0,C 180,E1 -16018.682,E2 -16018.682} C_VEL
LIN {X 0,Y 305.953,Z 250.376,A -85,B 0,C 180,E1 -16021.314,E2 -16021.314} C_VEL
LIN {X 0,Y 305.845,Z 250.387,A -85,B 0,C 180,E1 -16026.595,E2 -16026.595} C_VEL
LIN {X 0,Y 305.728,Z 250.403,A -85,B 0,C 180,E1 -16029.258,E2 -16029.258} C_VEL
LIN {X 0,Y 305.578,Z 250.424,A -85,B 0,C 180,E1 -16033.294,E2 -16033.294} C_VEL
LIN {X 0,Y 305.577,Z 250.428,A -85,B 0,C 180,E1 -16034.998,E2 -16034.998} C_VEL
LIN {X 0,Y 305.565,Z 251.645,A -85,B 0,C 180,E1 -16037.395,E2 -16037.395} C_VEL
LIN {X 0,Y 305.474,Z 253.432,A -85,B 0,C 180,E1 -16040.186,E2 -16040.186} C_VEL
LIN {X 0,Y 305.331,Z 255.344,A -85,B 0,C 180,E1 -16043.033,E2 -16043.033} C_VEL
LIN {X 0,Y 305.017,Z 258.469,A -85,B 0,C 180,E1 -16047.438,E2 -16047.438} C_VEL
LIN {X 0,Y 304.989,Z 258.679,A -85,B 0,C 180,E1 -16047.72,E2 -16047.72} C_VEL
LIN {X 0,Y 307.178,Z 264.569,A -85,B 0,C 180,E1 -16048.247,E2 -16048.247} C_VEL
LIN {X 0,Y 311.161,Z 275.508,A -85,B 0,C 180,E1 -16049.34,E2 -16049.34} C_VEL
LIN {X 0,Y 314.141,Z 286.592,A -85,B 0,C 180,E1 -16050.546,E2 -16050.546} C_VEL
LIN {X 0,Y 315.702,Z 294.981,A -85,B 0,C 180,E1 -16051.541,E2 -16051.541} C_VEL
LIN {X 0,Y 314.161,Z 305.766,A -85,B 0,C 180,E1 -16052.739,E2 -16052.739} C_VEL
LIN {X 0,Y 312.496,Z 316.274,A -85,B 0,C 180,E1 -16054.208,E2 -16054.208} C_VEL
LIN {X 0,Y 310.853,Z 325.827,A -85,B 0,C 180,E1 -16055.866,E2 -16055.866} C_VEL
LIN {X 0,Y 309.214,Z 334.216,A -85,B 0,C 180,E1 -16057.681,E2 -16057.681} C_VEL
LIN {X 0,Y 307.665,Z 341.881,A -85,B 0,C 180,E1 -16059.759,E2 -16059.759} C_VEL
LIN {X 0,Y 306.536,Z 347.465,A -85,B 0,C 180,E1 -16061.67,E2 -16061.67} C_VEL
LIN {X 0,Y 305.598,Z 351.963,A -85,B 0,C 180,E1 -16063.621,E2 -16063.621} C_VEL
LIN {X 0,Y 304.636,Z 356.304,A -85,B 0,C 180,E1 -16066.205,E2 -16066.205} C_VEL
LIN {X 0,Y 304.212,Z 358.291,A -85,B 0,C 180,E1 -16067.937,E2 -16067.937} C_VEL
LIN {X 0,Y 303.876,Z 359.579,A -85,B 0,C 180,E1 -16069.745,E2 -16069.745} C_VEL
LIN {X 0,Y 303.642,Z 360.175,A -85,B 0,C 180,E1 -16071.897,E2 -16071.897} C_VEL
LIN {X 0,Y 303.627,Z 359.707,A -85,B 0,C 180,E1 -16074.105,E2 -16074.105} C_VEL
LIN {X 0,Y 303.825,Z 358.077,A -85,B 0,C 180,E1 -16076.377,E2 -16076.377} C_VEL
LIN {X 0,Y 304.216,Z 355.088,A -85,B 0,C 180,E1 -16078.73,E2 -16078.73} C_VEL
LIN {X 0,Y 304.807,Z 350.468,A -85,B 0,C 180,E1 -16081.179,E2 -16081.179} C_VEL
LIN {X 0,Y 305.455,Z 345.358,A -85,B 0,C 180,E1 -16083.206,E2 -16083.206} C_VEL
LIN {X 0,Y 306.381,Z 338.815,A -85,B 0,C 180,E1 -16085.253,E2 -16085.253} C_VEL
LIN {X 0,Y 307.42,Z 331.285,A -85,B 0,C 180,E1 -16087.132,E2 -16087.132} C_VEL
LIN {X 0,Y 308.803,Z 321.592,A -85,B 0,C 180,E1 -16089.069,E2 -16089.069} C_VEL
LIN {X 0,Y 310.117,Z 311.777,A -85,B 0,C 180,E1 -16090.645,E2 -16090.645} C_VEL
LIN {X 0,Y 311.417,Z 300.451,A -85,B 0,C 180,E1 -16092.094,E2 -16092.094} C_VEL
LIN {X 0,Y 312.421,Z 290.068,A -85,B 0,C 180,E1 -16093.157,E2 -16093.157} C_VEL
LIN {X 0,Y 310.343,Z 279.092,A -85,B 0,C 180,E1 -16094.233,E2 -16094.233} C_VEL
LIN {X 0,Y 307.32,Z 266.723,A -85,B 0,C 180,E1 -16095.23,E2 -16095.23} C_VEL
LIN {X 0,Y 304.545,Z 256.272,A -85,B 0,C 180,E1 -16095.927,E2 -16095.927} C_VEL
LIN {X 0,Y 304.761,Z 252.178,A -85,B 0,C 180,E1 -16100.712,E2 -16100.712} C_VEL
LIN {X 0,Y 304.943,Z 250.85,A -85,B 0,C 180,E1 -16102.294,E2 -16102.294} C_VEL
LIN {X 0,Y 305.252,Z 250.459,A -85,B 0,C 180,E1 -16104.717,E2 -16104.717} C_VEL
LIN {X 0,Y 305.856,Z 250.384,A -85,B 0,C 180,E1 -16108.685,E2 -16108.685} C_VEL
LIN {X 0,Y 305.945,Z 250.377,A -85,B 0,C 180,E1 -16111.318,E2 -16111.318} C_VEL
LIN {X 0,Y 305.839,Z 250.386,A -85,B 0,C 180,E1 -16116.599,E2 -16116.599} C_VEL
LIN {X 0,Y 305.723,Z 250.404,A -85,B 0,C 180,E1 -16119.261,E2 -16119.261} C_VEL
LIN {X 0,Y 305.579,Z 250.421,A -85,B 0,C 180,E1 -16123.298,E2 -16123.298} C_VEL
LIN {X 0,Y 305.582,Z 250.418,A -85,B 0,C 180,E1 -16126.022,E2 -16126.022} C_VEL
LIN {X 0,Y 305.602,Z 250.417,A -85,B 0,C 180,E1 -16129.466,E2 -16129.466} C_VEL
LIN {X 0,Y 305.483,Z 250.435,A -85,B 0,C 180,E1 -16133.045,E2 -16133.045} C_VEL
LIN {X 0,Y 305.545,Z 250.424,A -85,B 0,C 180,E1 -16136.232,E2 -16136.232} C_VEL
LIN {X 0,Y 305.487,Z 250.433,A -85,B 0,C 180,E1 -16139.052,E2 -16139.052} C_VEL
LIN {X 0,Y 305.457,Z 250.433,A -85,B 0,C 180,E1 -16143.519,E2 -16143.519} C_VEL
LIN {X 0,Y 305.49,Z 250.434,A -85,B 0,C 180,E1 -16146.739,E2 -16146.739} C_VEL
LIN {X 0,Y 305.479,Z 250.435,A -85,B 0,C 180,E1 -16150.609,E2 -16150.609} C_VEL
LIN {X 0,Y 305.488,Z 250.429,A -85,B 0,C 180,E1 -16153.646,E2 -16153.646} C_VEL
LIN {X 0,Y 305.494,Z 250.428,A -85,B 0,C 180,E1 -16157.408,E2 -16157.408} C_VEL
LIN {X 0,Y 305.516,Z 250.425,A -85,B 0,C 180,E1 -16161.607,E2 -16161.607} C_VEL
LIN {X 0,Y 305.461,Z 250.43,A -85,B 0,C 180,E1 -16164.89,E2 -16164.89} C_VEL
LIN {X 0,Y 305.449,Z 250.438,A -85,B 0,C 180,E1 -16168.358,E2 -16168.358} C_VEL
LIN {X 0,Y 305.513,Z 250.426,A -85,B 0,C 180,E1 -16171.116,E2 -16171.116} C_VEL
LIN {X 0,Y 305.572,Z 250.423,A -85,B 0,C 180,E1 -16174.091,E2 -16174.091} C_VEL
LIN {X 0,Y 305.503,Z 250.427,A -85,B 0,C 180,E1 -16178.406,E2 -16178.406} C_VEL
LIN {X 0,Y 305.571,Z 250.414,A -85,B 0,C 180,E1 -16181.608,E2 -16181.608} C_VEL
LIN {X 0,Y 305.653,Z 250.409,A -85,B 0,C 180,E1 -16185.352,E2 -16185.352} C_VEL
LIN {X 0,Y 305.581,Z 250.417,A -85,B 0,C 180,E1 -16187.341,E2 -16187.341} C_VEL
LIN {X 0,Y 304.931,Z 250.502,A -85,B 0,C 180,E1 -16188.443,E2 -16188.443} C_VEL
LIN {X 0,Y 302.118,Z 250.85,A -85,B 0,C 180,E1 -16190.239,E2 -16190.239} C_VEL
LIN {X 0,Y 299.77,Z 251.143,A -85,B 0,C 180,E1 -16191.696,E2 -16191.696} C_VEL
LIN {X 0,Y 298.822,Z 251.257,A -85,B 0,C 180,E1 -16192.824,E2 -16192.824} C_VEL
LIN {X 0,Y 298.777,Z 251.262,A -85,B 0,C 180,E1 -16193.205,E2 -16193.205} C_VEL
LIN {X 0,Y 298.841,Z 251.257,A -85,B 0,C 180,E1 -16197.306,E2 -16197.306} C_VEL
LIN {X 0,Y 299.002,Z 251.24,A -85,B 0,C 180,E1 -16200.002,E2 -16200.002} C_VEL
LIN {X 0,Y 298.839,Z 251.257,A -85,B 0,C 180,E1 -16202.698,E2 -16202.698} C_VEL
LIN {X 0,Y 298.764,Z 251.264,A -85,B 0,C 180,E1 -16206.757,E2 -16206.757} C_VEL
LIN {X 0,Y 298.634,Z 251.284,A -85,B 0,C 180,E1 -16209.484,E2 -16209.484} C_VEL
LIN {X 0,Y 298.561,Z 251.297,A -85,B 0,C 180,E1 -16213.617,E2 -16213.617} C_VEL
LIN {X 0,Y 298.558,Z 251.292,A -85,B 0,C 180,E1 -16216.41,E2 -16216.41} C_VEL
LIN {X 0,Y 298.521,Z 251.299,A -85,B 0,C 180,E1 -16219.656,E2 -16219.656} C_VEL
LIN {X 0,Y 298.467,Z 251.307,A -85,B 0,C 180,E1 -16223.599,E2 -16223.599} C_VEL
LIN {X 0,Y 298.495,Z 251.3,A -85,B 0,C 180,E1 -16226.576,E2 -16226.576} C_VEL
LIN {X 0,Y 298.427,Z 251.311,A -85,B 0,C 180,E1 -16229.642,E2 -16229.642} C_VEL
LIN {X 0,Y 298.405,Z 251.314,A -85,B 0,C 180,E1 -16232.801,E2 -16232.801} C_VEL
LIN {X 0,Y 298.454,Z 251.308,A -85,B 0,C 180,E1 -16236.807,E2 -16236.807} C_VEL
LIN {X 0,Y 298.421,Z 251.314,A -85,B 0,C 180,E1 -16241.258,E2 -16241.258} C_VEL
LIN {X 0,Y 298.483,Z 251.524,A -85,B 0,C 180,E1 -16242.378,E2 -16242.378} C_VEL
LIN {X 0,Y 299.557,Z 257.508,A -85,B 0,C 180,E1 -16247.125,E2 -16247.125} C_VEL
LIN {X 0,Y 300.408,Z 262.525,A -85,B 0,C 180,E1 -16250.826,E2 -16250.826} C_VEL
LIN {X 0,Y 300.751,Z 266.25,A -85,B 0,C 180,E1 -16253.442,E2 -16253.442} C_VEL
LIN {X 0,Y 300.032,Z 271.041,A -85,B 0,C 180,E1 -16256.599,E2 -16256.599} C_VEL
LIN {X 0,Y 298.9,Z 278.25,A -85,B 0,C 180,E1 -16261.182,E2 -16261.182} C_VEL
LIN {X 0,Y 297.982,Z 285.406,A -85,B 0,C 180,E1 -16265.621,E2 -16265.621} C_VEL
LIN {X 0,Y 297.798,Z 287.028,A -85,B 0,C 180,E1 -16266.614,E2 -16266.614} C_VEL
LIN {X 0,Y 300.176,Z 300.782,A -85,B 0,C 180,E1 -16267.393,E2 -16267.393} C_VEL
LIN {X 0,Y 301.922,Z 314.372,A -85,B 0,C 180,E1 -16268.43,E2 -16268.43} C_VEL
LIN {X 0,Y 303.011,Z 326.881,A -85,B 0,C 180,E1 -16269.639,E2 -16269.639} C_VEL
LIN {X 0,Y 303.23,Z 334.627,A -85,B 0,C 180,E1 -16270.537,E2 -16270.537} C_VEL
LIN {X 0,Y 301.814,Z 344.771,A -85,B 0,C 180,E1 -16271.852,E2 -16271.852} C_VEL
LIN {X 0,Y 300.546,Z 354.342,A -85,B 0,C 180,E1 -16273.388,E2 -16273.388} C_VEL
LIN {X 0,Y 299.46,Z 362.717,A -85,B 0,C 180,E1 -16275.038,E2 -16275.038} C_VEL
LIN {X 0,Y 298.318,Z 371.049,A -85,B 0,C 180,E1 -16277.066,E2 -16277.066} C_VEL
LIN {X 0,Y 297.44,Z 377.758,A -85,B 0,C 180,E1 -16279.103,E2 -16279.103} C_VEL
LIN {X 0,Y 296.972,Z 383.111,A -85,B 0,C 180,E1 -16281.15,E2 -16281.15} C_VEL
LIN {X 0,Y 296.737,Z 387.263,A -85,B 0,C 180,E1 -16283.198,E2 -16283.198} C_VEL
LIN {X 0,Y 296.647,Z 389.433,A -85,B 0,C 180,E1 -16284.561,E2 -16284.561} C_VEL
LIN {X 0,Y 296.684,Z 391.122,A -85,B 0,C 180,E1 -16285.923,E2 -16285.923} C_VEL
LIN {X 0,Y 296.664,Z 392.39,A -85,B 0,C 180,E1 -16287.283,E2 -16287.283} C_VEL
LIN {X 0,Y 296.733,Z 393.256,A -85,B 0,C 180,E1 -16288.641,E2 -16288.641} C_VEL
LIN {X 0,Y 296.812,Z 393.685,A -85,B 0,C 180,E1 -16289.999,E2 -16289.999} C_VEL
LIN {X 0,Y 296.692,Z 393.681,A -85,B 0,C 180,E1 -16291.356,E2 -16291.356} C_VEL
LIN {X 0,Y 296.637,Z 393.286,A -85,B 0,C 180,E1 -16292.715,E2 -16292.715} C_VEL
LIN {X 0,Y 296.619,Z 392.501,A -85,B 0,C 180,E1 -16294.075,E2 -16294.075} C_VEL
LIN {X 0,Y 296.594,Z 391.114,A -85,B 0,C 180,E1 -16295.591,E2 -16295.591} C_VEL
LIN {X 0,Y 296.86,Z 387.579,A -85,B 0,C 180,E1 -16298.165,E2 -16298.165} C_VEL
LIN {X 0,Y 297.31,Z 383.621,A -85,B 0,C 180,E1 -16300.211,E2 -16300.211} C_VEL
LIN {X 0,Y 298.021,Z 378.549,A -85,B 0,C 180,E1 -16302.252,E2 -16302.252} C_VEL
LIN {X 0,Y 299.294,Z 372.226,A -85,B 0,C 180,E1 -16304.273,E2 -16304.273} C_VEL
LIN {X 0,Y 300.744,Z 364.394,A -85,B 0,C 180,E1 -16306.284,E2 -16306.284} C_VEL
LIN {X 0,Y 302.43,Z 354.671,A -85,B 0,C 180,E1 -16308.282,E2 -16308.282} C_VEL
LIN {X 0,Y 304.346,Z 344.73,A -85,B 0,C 180,E1 -16309.912,E2 -16309.912} C_VEL
LIN {X 0,Y 305.786,Z 336.308,A -85,B 0,C 180,E1 -16311.044,E2 -16311.044} C_VEL
LIN {X 0,Y 305.811,Z 326.608,A -85,B 0,C 180,E1 -16312.252,E2 -16312.252} C_VEL
LIN {X 0,Y 304.855,Z 314.651,A -85,B 0,C 180,E1 -16313.554,E2 -16313.554} C_VEL
LIN {X 0,Y 302.838,Z 302.036,A -85,B 0,C 180,E1 -16314.731,E2 -16314.731} C_VEL
LIN {X 0,Y 299.449,Z 288.241,A -85,B 0,C 180,E1 -16315.867,E2 -16315.867} C_VEL
LIN {X 0,Y 298.508,Z 284.57,A -85,B 0,C 180,E1 -16316.157,E2 -16316.157} C_VEL
LIN {X 0,Y 299.603,Z 277.039,A -85,B 0,C 180,E1 -16321.067,E2 -16321.067} C_VEL
LIN {X 0,Y 300.848,Z 271.084,A -85,B 0,C 180,E1 -16325.15,E2 -16325.15} C_VEL
LIN {X 0,Y 301.214,Z 267.9,A -85,B 0,C 180,E1 -16327.503,E2 -16327.503} C_VEL
LIN {X 0,Y 300.904,Z 265.323,A -85,B 0,C 180,E1 -16329.576,E2 -16329.576} C_VEL
LIN {X 0,Y 300.107,Z 260.887,A -85,B 0,C 180,E1 -16333.448,E2 -16333.448} C_VEL
LIN {X 0,Y 299.403,Z 257.143,A -85,B 0,C 180,E1 -16337.097,E2 -16337.097} C_VEL
LIN {X 0,Y 298.837,Z 253.678,A -85,B 0,C 180,E1 -16340.901,E2 -16340.901} C_VEL
LIN {X 0,Y 298.42,Z 251.315,A -85,B 0,C 180,E1 -16343.928,E2 -16343.928} C_VEL
LIN {X 0,Y 298.394,Z 251.319,A -85,B 0,C 180,E1 -16347.981,E2 -16347.981} C_VEL
LIN {X 0,Y 298.461,Z 251.309,A -85,B 0,C 180,E1 -16351.902,E2 -16351.902} C_VEL
LIN {X 0,Y 298.483,Z 251.306,A -85,B 0,C 180,E1 -16354.922,E2 -16354.922} C_VEL
LIN {X 0,Y 298.447,Z 251.311,A -85,B 0,C 180,E1 -16359.313,E2 -16359.313} C_VEL
LIN {X 0,Y 298.534,Z 251.299,A -85,B 0,C 180,E1 -16362.177,E2 -16362.177} C_VEL
LIN {X 0,Y 298.589,Z 251.293,A -85,B 0,C 180,E1 -16364.993,E2 -16364.993} C_VEL
LIN {X 0,Y 298.591,Z 251.292,A -85,B 0,C 180,E1 -16369.145,E2 -16369.145} C_VEL
LIN {X 0,Y 298.753,Z 251.272,A -85,B 0,C 180,E1 -16371.884,E2 -16371.884} C_VEL
LIN {X 0,Y 298.656,Z 251.284,A -85,B 0,C 180,E1 -16374.597,E2 -16374.597} C_VEL
LIN {X 0,Y 298.918,Z 251.252,A -85,B 0,C 180,E1 -16378.651,E2 -16378.651} C_VEL
LIN {X 0,Y 298.919,Z 251.252,A -85,B 0,C 180,E1 -16381.345,E2 -16381.345} C_VEL
LIN {X 0,Y 298.79,Z 251.266,A -85,B 0,C 180,E1 -16386.752,E2 -16386.752} C_VEL
LIN {X 0,Y 298.673,Z 251.283,A -85,B 0,C 180,E1 -16389.478,E2 -16389.478} C_VEL
LIN {X 0,Y 298.533,Z 251.303,A -85,B 0,C 180,E1 -16393.614,E2 -16393.614} C_VEL
LIN {X 0,Y 298.544,Z 251.561,A -85,B 0,C 180,E1 -16395.17,E2 -16395.17} C_VEL
LIN {X 0,Y 298.548,Z 253.96,A -85,B 0,C 180,E1 -16399.24,E2 -16399.24} C_VEL
LIN {X 0,Y 298.252,Z 256.849,A -85,B 0,C 180,E1 -16403.612,E2 -16403.612} C_VEL
LIN {X 0,Y 298.015,Z 259.225,A -85,B 0,C 180,E1 -16406.948,E2 -16406.948} C_VEL
LIN {X 0,Y 299.104,Z 262.253,A -85,B 0,C 180,E1 -16407.22,E2 -16407.22} C_VEL
LIN {X 0,Y 303.811,Z 274.36,A -85,B 0,C 180,E1 -16408.476,E2 -16408.476} C_VEL
LIN {X 0,Y 307.127,Z 285.993,A -85,B 0,C 180,E1 -16409.784,E2 -16409.784} C_VEL
LIN {X 0,Y 309.045,Z 295.543,A -85,B 0,C 180,E1 -16410.962,E2 -16410.962} C_VEL
LIN {X 0,Y 308.807,Z 299.163,A -85,B 0,C 180,E1 -16411.37,E2 -16411.37} C_VEL
LIN {X 0,Y 306.987,Z 310.448,A -85,B 0,C 180,E1 -16412.754,E2 -16412.754} C_VEL
LIN {X 0,Y 305.181,Z 321.065,A -85,B 0,C 180,E1 -16414.42,E2 -16414.42} C_VEL
LIN {X 0,Y 303.404,Z 330.416,A -85,B 0,C 180,E1 -16416.256,E2 -16416.256} C_VEL
LIN {X 0,Y 301.756,Z 337.902,A -85,B 0,C 180,E1 -16418.08,E2 -16418.08} C_VEL
LIN {X 0,Y 300.235,Z 345.23,A -85,B 0,C 180,E1 -16420.338,E2 -16420.338} C_VEL
LIN {X 0,Y 299.167,Z 350.087,A -85,B 0,C 180,E1 -16422.238,E2 -16422.238} C_VEL
LIN {X 0,Y 298.315,Z 353.789,A -85,B 0,C 180,E1 -16424.067,E2 -16424.067} C_VEL
LIN {X 0,Y 297.402,Z 357.697,A -85,B 0,C 180,E1 -16426.742,E2 -16426.742} C_VEL
LIN {X 0,Y 296.859,Z 359.809,A -85,B 0,C 180,E1 -16429.248,E2 -16429.248} C_VEL
LIN {X 0,Y 296.563,Z 360.595,A -85,B 0,C 180,E1 -16431.966,E2 -16431.966} C_VEL
LIN {X 0,Y 296.52,Z 360.253,A -85,B 0,C 180,E1 -16433.688,E2 -16433.688} C_VEL
LIN {X 0,Y 296.678,Z 358.8,A -85,B 0,C 180,E1 -16436.003,E2 -16436.003} C_VEL
LIN {X 0,Y 297.102,Z 355.71,A -85,B 0,C 180,E1 -16438.642,E2 -16438.642} C_VEL
LIN {X 0,Y 297.647,Z 351.742,A -85,B 0,C 180,E1 -16440.878,E2 -16440.878} C_VEL
LIN {X 0,Y 298.292,Z 346.66,A -85,B 0,C 180,E1 -16443.03,E2 -16443.03} C_VEL
LIN {X 0,Y 299.313,Z 339.755,A -85,B 0,C 180,E1 -16445.297,E2 -16445.297} C_VEL
LIN {X 0,Y 300.404,Z 332.06,A -85,B 0,C 180,E1 -16447.294,E2 -16447.294} C_VEL
LIN {X 0,Y 301.65,Z 323.664,A -85,B 0,C 180,E1 -16449.048,E2 -16449.048} C_VEL
LIN {X 0,Y 302.99,Z 313.954,A -85,B 0,C 180,E1 -16450.7,E2 -16450.7} C_VEL
LIN {X 0,Y 304.287,Z 303.938,A -85,B 0,C 180,E1 -16452.081,E2 -16452.081} C_VEL
LIN {X 0,Y 305.441,Z 293.092,A -85,B 0,C 180,E1 -16453.286,E2 -16453.286} C_VEL
LIN {X 0,Y 305.399,Z 289.704,A -85,B 0,C 180,E1 -16453.628,E2 -16453.628} C_VEL
LIN {X 0,Y 303.048,Z 278.056,A -85,B 0,C 180,E1 -16454.783,E2 -16454.783} C_VEL
LIN {X 0,Y 299.815,Z 265.241,A -85,B 0,C 180,E1 -16455.808,E2 -16455.808} C_VEL
LIN {X 0,Y 297.492,Z 256.663,A -85,B 0,C 180,E1 -16456.38,E2 -16456.38} C_VEL
LIN {X 0,Y 297.686,Z 253.202,A -85,B 0,C 180,E1 -16460.489,E2 -16460.489} C_VEL
